// TwinCAT 3 PLC project TestHarnessCore
// Title: TestHarnessCore
// Company: None
// ProjectVersion: 0.0.11
// ProgramVersion: 3.1.4026.24
// libraries:
//   Tc2_Standard, * (Beckhoff Automation GmbH)
//   Tc2_System, * (Beckhoff Automation GmbH)
//   Tc2_Utilities, * (Beckhoff Automation GmbH)
//   Tc3_EventLogger, * (Beckhoff Automation GmbH)
//   Tc3_JsonXml, * (Beckhoff Automation GmbH)
// project tree:
//   DUTs/ E_FailureKind.TcDUT, E_PhaseOutcome.TcDUT, E_RegistrationFault.TcDUT, E_RunOutcome.TcDUT, E_RunPhase.TcDUT, E_TestStatus.TcDUT, ST_CompareResult.TcDUT, ST_NumericValue.TcDUT, ST_TestBudget.TcDUT, ST_TestBudgets.TcDUT, ST_TestRunStatus.TcDUT, ST_TestSlot.TcDUT
//   Interfaces/ I_TestCyclic.TcIO, I_Labelled.TcIO, I_Test.TcIO, I_TestAssertions.TcIO, I_TestConfiguration.TcIO, I_TestDefaults.TcIO, I_TestDetailSink.TcIO, I_TestExecution.TcIO, I_TestJournalSet.TcIO, I_TestLocation.TcIO, I_TestOutcome.TcIO, I_TestRegistrar.TcIO, I_TestReporter.TcIO, I_TestReRun.TcIO, I_TestRegistration.TcIO, I_TestRoster.TcIO, I_TestRunRegistration.TcIO, I_TestRunStatus.TcIO, I_TestSetup.TcIO, I_TestSuite.TcIO, I_TestTeardown.TcIO, I_TestTiming.TcIO
//   Parameters/ TestHarnessParameter.TcGVL
//   POUs/ TestArbiter.TcPOU, TestDeadline.TcPOU, TestEventReporter.TcPOU, TestJournal.TcPOU, TestJUnitReporter.TcPOU, TestLogReporter.TcPOU, TestRegistry.TcPOU, TestReporterFanout.TcPOU, TestRun.TcPOU, TestRunner.TcPOU, TestRunTally.TcPOU, TestStopwatch.TcPOU, TestSuite.TcPOU, TestSummaryLine.TcPOU, TestTimeoutDiagnostic.TcPOU, TestValueAsLReal.TcPOU, TestValueBrief.TcPOU, TestValueCompare.TcPOU, TestValueIsFloat.TcPOU, TestValueIsText.TcPOU, TestValueString.TcPOU, TestVerdict.TcPOU
//   Project Information/ F_GetCompany.TcPOU, F_GetTitle.TcPOU, F_GetVersion.TcPOU
//   Version/ Global_Version.TcGVL
// real-time tasks:
//   TASK PlcTask: cycle T#10ms, priority 20, ADS port 350

// ---- DUTs/E_FailureKind.TcDUT
// Why a test did not pass. Carried in the result document's failure 'type'

// attribute. A single hardcoded 'AssertionError' for everything makes that field

// making a machine-readable field useless.

//

// Keeping the kind here frees the 80-character summary from repeating it, and

// gives CI something to group by.
{attribute 'qualified_only'}
{attribute 'strict'}
TYPE E_FailureKind : (
		None		  := 0,
		ValueMismatch := 1,
		TypeMismatch  := 2,
		SizeMismatch  := 3,
		Timeout		  := 4,
		Aborted		  := 5,
		Environment	  := 6
	) DINT;
END_TYPE

// ---- DUTs/E_PhaseOutcome.TcDUT
// What one scan of TestRunner.Advance did.

//

// TeardownOverran is separate from Finished because the two need different action

// from the caller, and the runner cannot take it: the suite holds the reporters.

// The test's VERDICT is unaffected either way - a passing test whose cleanup hung

// still proved the code correct - but the run must go red, and only the suite can

// say so.
{attribute 'qualified_only'}
{attribute 'strict'}
TYPE E_PhaseOutcome : (
		// Nothing is loaded. Load a test before advancing.
		Idle := 0,
		// Still working. Call again next scan.
		Running := 1,
		// Terminal, cleanly. The verdict is in the journal.
		Finished := 2,
		// Terminal, but teardown hit its deadline and was abandoned. On a rig this may

		// mean an axis left powered. Raise a framework error; do not touch the verdict.
		TeardownOverran := 3
	) DINT;
END_TYPE

// ---- DUTs/E_RegistrationFault.TcDUT
// Why a registration was refused. None means it was accepted.

//

// Distinct causes rather than one BOOL, because each needs a different action from

// whoever reads the report: resize the suite, rename a test, supply the missing

// argument, move the call earlier. A rejected registration is never silent - a

// test that failed to register would otherwise vanish from the results and CI

// would see fewer passes rather than a failure.
{attribute 'qualified_only'}
{attribute 'strict'}
TYPE E_RegistrationFault : (
		None := 0,
		// No free slot. A sizing error: raise the generic argument on the declaration,

		// or split the suite.
		Full := 1,
		// The label is already used in this suite. Labels are the key CI trend history

		// is built on, so two tests cannot share one.
		DuplicateLabel := 2,
		// No label supplied. Usually a missing argument at the call site.
		EmptyLabel := 3,
		// No test supplied. Its own cause rather than folded into EmptyLabel, because

		// reporting the wrong one sends the reader to the wrong argument.
		NoTest := 5,
		// The suite has already been enabled. Registration closes then and a re-run does

		// not reopen it: a re-run re-executes the registered set, it does not redefine

		// it.
		Closed := 4
	) DINT;
END_TYPE

// ---- DUTs/E_RunOutcome.TcDUT
// The aggregate state of a suite, or of a sequencer aggregating suites.

//

// The members mirror E_TestStatus but the type is separate on purpose: a run

// outcome is not a test verdict, and a single type would invite passing one where

// the other is meant.

//

// Aggregation rules, applied in order:

//   any Errored          -> Errored     (the run could not be trusted)

//   any Failed           -> Failed

//   all Skipped          -> Skipped

//   otherwise            -> Passed

//

// Errored outranks Failed because a framework or environment problem casts doubt

// on every other result in the run.
{attribute 'qualified_only'}
{attribute 'strict'}
TYPE E_RunOutcome : (
		NotStarted := 0,
		Running	   := 1,
		Passed	   := 2,
		Failed	   := 3,
		Errored	   := 4,
		Skipped	   := 5
	) DINT;
END_TYPE

// ---- DUTs/E_RunPhase.TcDUT
// Which phase of one test the runner is in. Internal to TestRunner - nothing

// outside it needs to know, and exposing it would invite someone to branch on it.
{attribute 'qualified_only'}
{attribute 'strict'}
TYPE E_RunPhase : (
		Idle	 := 0,
		Setup	 := 1,
		Body	 := 2,
		Teardown := 3
	) DINT;
END_TYPE

// ---- DUTs/E_TestStatus.TcDUT
// The state of a single test.

//

// Six members, each earned: the suite needs to know what to run next, the result

// document needs the four terminal values, and CI needs the last two kept out of

// the failure count.

//

// Errored is deliberately distinct from Failed. Failed means an assertion did not

// hold - the code under test was shown to be wrong. Errored means the test could

// not run: a precondition was absent, a target was unreachable. Conflating them

// sends whoever reads the report hunting a defect that is not there.

//

// The order is NOT load-bearing. Ask IsTerminal() rather than comparing ordinals,

// so that adding a member later is not a breaking change.
{attribute 'qualified_only'}
{attribute 'strict'}
TYPE E_TestStatus : (
		NotStarted := 0,
		Running	   := 1,
		Passed	   := 2,
		Failed	   := 3,
		Errored	   := 4,
		Skipped	   := 5
	) DINT;
END_TYPE

// ---- DUTs/ST_CompareResult.TcDUT
// What TestValueCompare found. A value, not a verdict - nothing is recorded until

// a caller decides to record it.
TYPE ST_CompareResult :
	STRUCT
		IsEqual : BOOL;
		// Why not, when IsEqual is FALSE. None when it is TRUE.
		Kind : E_FailureKind;
		// The composed one-line form, for the summary. Each value in it is shortened to

		// a per-value budget, because both of them plus the surrounding words cannot fit

		// in 255 characters and CONCAT cannot build a longer string than that.

		//

		// Never the author's message - the comparison knows nothing about intent.
		Diagnostic : T_MaxString;
		// The values as rendered, in full, each in its own field so neither is cut by

		// the other. Empty when IsEqual, and empty for a failure that has no two values

		// to show - a size mismatch, a type mismatch.

		//

		// A value whose rendering exceeds 255 characters is still cut here. Comparing

		// something that long is what AssertBufferEqual is for.
		Expected : T_MaxString;
		Actual	 : T_MaxString;
	END_STRUCT
END_TYPE

// ---- DUTs/ST_NumericValue.TcDUT
// A number recovered from an ANY, and whether one was there to recover.

//

// IsNumeric is FALSE for strings, structs, arrays and anything else with no

// ordering. Value is 0.0 in that case and must not be read.

//

// This is a return type rather than an output parameter because an output binds

// with => and never positionally, so a caller writing TestValueAsLReal(V, Ok)

// would bind Ok to an input and never see the flag.
{attribute 'pack_mode' := '1'}
TYPE ST_NumericValue :
	STRUCT
		IsNumeric : BOOL;
		Value	  : LREAL;
	END_STRUCT
END_TYPE

// ---- DUTs/ST_TestBudget.TcDUT
// A deadline for one phase of one test, in both units.

//

// The two units are tracked independently. A test naming its own wall-clock

// budget still inherits the suite's scan budget, and the reverse.

//

// ZERO DISABLES. A budget of zero means no deadline for that unit, which is why

// "not specified" needs its own flag and cannot be inferred from the value. The

// two meanings are different and both are needed: a long-running rig test may

// legitimately want no scan budget at all.
TYPE ST_TestBudget :
	STRUCT
		// Scan budget. The reproducible unit - prefer it. Zero disables.
		Cycles : UDINT;
		// FALSE means "not specified here": inherit the suite default at registration,

		// or leave the existing default unchanged when setting defaults.
		IsCyclesSet : BOOL;
		// Wall-clock budget. Varies with jitter across targets. Zero disables.
		Timeout		 : TIME;
		IsTimeoutSet : BOOL;
	END_STRUCT
END_TYPE

// ---- DUTs/ST_TestBudgets.TcDUT
// The three deadlines a test can have, one per phase.

//

// Three rather than one because the phases are not the same kind of work. Setup

// may legitimately be slow - waiting for hardware to answer. Teardown should not

// be: stopping motion and dropping power is near-immediate, and if it is not,

// that is the fault being detected. Giving teardown the body's budget would leave

// an axis powered for the whole of it.

//

// An untouched instance specifies nothing and inherits every suite default, which

// is what the great majority of registrations want. Declare one in the

// composition root and pass it to every Register that has nothing to say.
TYPE ST_TestBudgets :
	STRUCT
		// Bounds I_TestSetup.Setup. Ignored by a test that does not implement it.
		Setup : ST_TestBudget;
		// Bounds I_Test.Run. This is the original deadline, from when a test grew from

		// one scan to many.
		Body : ST_TestBudget;
		// Bounds I_TestTeardown.Teardown. Overrunning it does NOT change the test's

		// verdict - a passing test whose cleanup hung still proved the code correct -

		// but it is reported as a framework error and turns the run red.
		Teardown : ST_TestBudget;
	END_STRUCT
END_TYPE

// ---- DUTs/ST_TestRunStatus.TcDUT
// The same figures I_TestRunStatus exposes, as a plain struct.

//

// Published alongside the interface so ADS, TwinCAT HMI and OPC UA read the run

// as ordinary symbols without RPC. That is the portable path and the one CI

// polls: an interface is not reachable from outside the PLC, and a design that

// exposed neither - the only signals were a file appearing on disk and a line in

// a log, both of which have to be scraped.
TYPE ST_TestRunStatus :
	STRUCT
		Label	: T_MaxString;
		Outcome : E_RunOutcome;
		// Reached a terminal state - NOT "ran everything". A skipped suite is complete.
		IsComplete : BOOL;
		// Once complete, Passed + Failed + Errored + Skipped equals TestCount.
		TestCount	: UDINT;
		PassedCount : UDINT;
		FailedCount : UDINT;
		// Tests that could not run, plus framework errors. Kept apart from FailedCount

		// because a build should react differently: a failure means the code is wrong,

		// an error means the run cannot be trusted.
		ErrorCount	  : UDINT;
		SkippedCount  : UDINT;
		TotalDuration : LREAL;
	END_STRUCT
END_TYPE

// ---- DUTs/ST_TestSlot.TcDUT
// One registered test, as the registry holds it.

//

// The three optional hooks are resolved ONCE, by __QUERYINTERFACE at registration,

// and stored. Querying them per scan would put an interface lookup in cyclic code

// for a result that cannot change - the instance a slot points at is fixed for the

// life of the run.

//

// A hook the test does not implement is a null reference, which is the whole test:

// no base class, no empty method bodies, no flags to keep in step with reality.
TYPE ST_TestSlot :
	STRUCT
		// Null in a slot that was never claimed. This is the "is there a test here"

		// question - never an index compared against a count.
		Test : I_Test;
		// Where this slot sits in registration order, so a holder of the slot can reach

		// the matching journal without carrying a second value alongside it. -1 in an

		// unclaimed slot.
		Index : DINT := -1;
		Label : T_MaxString;
		// Null unless the test implements the corresponding optional interface.
		Setup	 : I_TestSetup;
		Teardown : I_TestTeardown;
		Location : I_TestLocation;
	END_STRUCT
END_TYPE

// ---- Parameters/TestHarnessParameter.TcGVL
// Dials a referencing project can turn from the Library Manager, without editing

// this library.

//

// Everything here is a DEFAULT, not a limit. Capacity is overridable per instance

// as well - TestRegistry<20> - so this is the value a declaration inherits when it

// says nothing.
{attribute 'qualified_only'}
VAR_GLOBAL CONSTANT
	// Tests a suite can hold. Every slot costs its journal whether used or not, so

	// prefer several small suites to one large one.

	//

	// Must be at least 1: ARRAY[0..Capacity - 1] with zero is a compile error, and

	// that is the right outcome. Clamping a zero to one slot would be the same class

	// of silent surprise this library exists to remove.
	Capacity : UDINT := 10;

	// Sinks a suite or sequencer can hold. Not a generic argument: a project

	// attaches the same set of sinks to every suite it owns, so per-instance

	// variation would cost every declaration site a second argument to buy nothing.
	ReporterCapacity : UDINT := 4;

	// Suites a TestRun can hold. A project usually has a handful - unit, motion,

	// I/O - so this is small on purpose, and overridable per instance as a generic

	// argument like Capacity.
	SuiteCapacity : UDINT := 8;

	// Scans a suite may go WITHOUT COMPLETING A TEST before the run abandons it.

	//

	// Not scans since the suite started - that would fire on a slow suite rather

	// than a stuck one. A rig suite waiting on hardware can sit for minutes and be

	// perfectly healthy, but it still finishes its tests one at a time; a stalled one

	// finishes none.

	//

	// Generous on purpose. This is a BACKSTOP: per-test deadlines already bound

	// every test that did not disable them, so the only things left for this to catch

	// are a framework defect and a test that turned its own deadlines off and hung.

	// A single legitimate test that takes longer than this needs it raised.

	//

	// Zero disables it, like every other deadline in this library.
	SuiteWatchdogCycles : UDINT := 60000;
END_VAR

// ---- Version/Global_Version.TcGVL
{attribute 'TcGenerated'}
{attribute 'no-analysis'}
{attribute 'linkalways'}
// This function has been automatically generated from the project information.
VAR_GLOBAL CONSTANT
	{attribute 'const_non_replaced'}
	stLibVersion_TestHarnessCore : ST_LibVersion := (iMajor := 0, iMinor := 0, iBuild := 11, iRevision := 0, nFlags := 0, sVersion := '0.0.11');
END_VAR

// ---- Interfaces/I_TestCyclic.TcIO
// Something with per-scan work.

//

// The bottom of the stack, with IQueryInterface beneath it. Every interface in

// this library reaches IQueryInterface through its own root, so any reference can

// be queried for any other role it plays.
INTERFACE I_TestCyclic EXTENDS __SYSTEM.IQueryInterface

// Called every scan, unconditionally, by whatever owns this object.

//

// The name is the contract. An Execute input would mean a trigger; an Enable

// input would mean held-while-wanted; CyclicLogic means there is no gating

// condition and the caller must not invent one.
METHOD CyclicLogic
END_METHOD

END_INTERFACE

// ---- Interfaces/I_Labelled.TcIO
// Something that carries a human-readable name.

//

// Extracted because a suite needs a label in two unrelated roles - as the thing

// the sequencer drives, and as the thing an observer reads counts from - and

// declaring it twice would let the two drift apart.
INTERFACE I_Labelled EXTENDS __SYSTEM.IQueryInterface

// The name that appears in results. Stable across renames of the underlying

// instance, because it is supplied rather than derived.
PROPERTY Label : T_MaxString
GET
END_GET
END_PROPERTY

END_INTERFACE

// ---- Interfaces/I_Test.TcIO
// A test. Implemented by test code you write - never by the code under test.

//

// One method is the entire framework contract for a test author.

//

// Reaches IQueryInterface so the suite can ask, at registration, whether a test

// also implements I_TestSetup, I_TestTeardown or I_TestLocation. Those three are

// optional and independent: implement none, one, or all, with no empty bodies for

// the ones you do not want. They do not share a base interface because they would

// have to share a method name, and a test implementing two would then collide.
INTERFACE I_Test EXTENDS __SYSTEM.IQueryInterface

// Called by the suite once per scan while this test is the active one, and never

// otherwise. There is no gate to check and no permission to ask: if you were

// called, run.

//

// Return TRUE when there is no more work. A single-scan test returns TRUE on its

// first call; a multi-scan test returns FALSE until its state machine finishes.

// The test declares completion - the framework never infers it from the checks,

// Without it a test can end at its first passing check and report

// green on work it never reached.

//

// Enable is held TRUE while the test should keep running. The suite drops it to

// abandon a test, on reset or re-run. On a falling edge the test returns its own

// state to its starting condition and returns TRUE; the value is otherwise

// ignored in that case.

//

// The verdict is not returned here. It is whatever the checks recorded through

// Test, and it belongs to the runner.
METHOD Run : BOOL
VAR_INPUT
	Enable : BOOL;
	Test   : I_TestAssertions;
END_VAR
END_METHOD

END_INTERFACE

// ---- Interfaces/I_TestAssertions.TcIO
// The handle a test body reports through: the verdict surface, the runner's

// timing, and the built-in comparisons.

//

// Handed to the test on every call. Never held, never stored.

//

// Everything here is a convenience over I_TestOutcome.RecordPass and

// RecordFailure. Domain helpers should take the narrower I_TestOutcome instead -

// they report, they do not need to compare.

//

// There is no WaitUntil. A test that is not finished returns FALSE from Run and is

// called again; waiting is the absence of returning TRUE.
INTERFACE I_TestAssertions EXTENDS I_TestOutcome, I_TestTiming

// As AssertMemEqual, but lengths are compared first and a mismatch is reported

// as SizeMismatch rather than as a difference at some offset.
METHOD AssertBufferEqual
VAR_INPUT
	pExpected	   : POINTER TO BYTE;
	ExpectedLength : UDINT;
	pActual		   : POINTER TO BYTE;
	ActualLength   : UDINT;
	Message		   : T_MaxString;
END_VAR
END_METHOD

// Asserts the test has COMPLETED no more than Cycles scans. Built on

// I_TestTiming.ElapsedCycles, so it needs no bookkeeping from the test.

//

// The scan in progress is not counted - see I_TestTiming.ElapsedCycles. A body

// checking this on its third call is asserting about the two scans that finished,

// not the three it has been called for. Assert it on the scan AFTER the work is

// done, which is where the answer is known anyway:

//

//   IF Sut.IsDone THEN

//       Test.AssertCompletedWithin(2, 'homing took too long');

//       Run := TRUE;

//   END_IF

//

// Opt-in, never a default. A scan budget is a real regression signal on a fixed

// target and noise across a matrix of them.
METHOD AssertCompletedWithin
VAR_INPUT
	Cycles	: UDINT;
	Message : T_MaxString;
END_VAR
END_METHOD

// Compares two values of the same type, including strings and enums.

//

// ANY binds only to an addressable variable. A literal, a property or an inlined

// constant will not compile, so both sides must be copied into variables first.

// A language constraint, not a choice.
METHOD AssertEqual
VAR_INPUT
	Expected : ANY;
	Actual	 : ANY;
	Message	 : T_MaxString;
END_VAR
END_METHOD

METHOD AssertFalse
VAR_INPUT
	Condition : BOOL;
	Message	  : T_MaxString;
END_VAR
END_METHOD

// Actual > Bound. Numeric types only. See AssertEqual on the ANY constraint.
METHOD AssertGreater
VAR_INPUT
	Actual	: ANY;
	Bound	: ANY;
	Message : T_MaxString;
END_VAR
END_METHOD

// Inclusive on both bounds.
METHOD AssertInRange
VAR_INPUT
	Actual	: LREAL;
	Minimum : LREAL;
	Maximum : LREAL;
	Message : T_MaxString;
END_VAR
END_METHOD

// Actual < Bound. Numeric types only. See AssertEqual on the ANY constraint.
METHOD AssertLess
VAR_INPUT
	Actual	: ANY;
	Bound	: ANY;
	Message : T_MaxString;
END_VAR
END_METHOD

// Byte comparison of two regions of equal length. Reports the offset of the

// first difference.
METHOD AssertMemEqual
VAR_INPUT
	pExpected : POINTER TO BYTE;
	pActual	  : POINTER TO BYTE;
	Length	  : UDINT;
	Message	  : T_MaxString;
END_VAR
END_METHOD

// ABSOLUTE tolerance: passes when |Expected - Actual| <= Tolerance.

//

// Tolerance carries the units of the value compared - millimetres, volts, counts.

// Its counterpart is AssertWithin, which takes a fraction instead.

//

// AssertEqual compares floats EXACTLY. Tolerance is never applied implicitly, so

// choosing it is visible at the call site.
METHOD AssertNear
VAR_INPUT
	Expected  : LREAL;
	Actual	  : LREAL;
	Tolerance : LREAL;
	Message	  : T_MaxString;
END_VAR
END_METHOD

// See AssertEqual on the ANY constraint.
METHOD AssertNotEqual
VAR_INPUT
	Expected : ANY;
	Actual	 : ANY;
	Message	 : T_MaxString;
END_VAR
END_METHOD

METHOD AssertTrue
VAR_INPUT
	Condition : BOOL;
	Message	  : T_MaxString;
END_VAR
END_METHOD

// RELATIVE tolerance: passes when |Expected - Actual| <= |Expected| * Fraction.

//

// Holds its meaning across magnitudes, which absolute tolerance does not. Near

// zero it collapses to exact equality - if zero is the expected value, use

// AssertNear.
METHOD AssertWithin
VAR_INPUT
	Expected : LREAL;
	Actual	 : LREAL;

	// Dimensionless. 0.001 is 0.1 per cent of Expected.
	Fraction : LREAL;
	Message	 : T_MaxString;
END_VAR
END_METHOD

END_INTERFACE

// ---- Interfaces/I_TestConfiguration.TcIO
// Startup configuration common to a suite and a sequencer: what it is called, and

// where its results go. Held by the composition root and nothing else.

//

// Shared by both because both implement I_TestRunStatus - so both carry a label -

// and both fan results out to sinks. The two suite-only faces stay separate:

// I_TestRegistration adds tests, I_TestDefaults sets deadline defaults, and a

// sequencer has neither.

//

// Everything here is set before the object is first enabled. Nothing on this

// interface is safe to call from cyclic code.
INTERFACE I_TestConfiguration EXTENDS __SYSTEM.IQueryInterface

// Attach a sink. Every reporter attached receives every result; there is no

// filtering here, because a sink that wants less can decide that for itself.

//

// Order of attachment is order of notification, which matters for one thing only:

// a sink that writes a file and a sink that raises an alarm should not be relied

// on to complete in any particular order relative to each other. If sequencing

// between two sinks matters, that is one sink wrapping two.

//

// Returns FALSE when the reporter list is full or the object is already running,

// and raises a framework error through the reporters ALREADY attached. That is

// not circular: the ones already there are exactly the ones that can still report

// it. A rejection with no reporters attached at all is silent, and is the reason

// ReporterCount exists.
METHOD AddReporter : BOOL
VAR_INPUT
	Reporter : I_TestReporter;
END_VAR
END_METHOD

// Assert this in CI against an expected number.

//

// A reporter that silently stops being attached takes its output with it - the

// result file simply never appears - and the pipeline reads that as a broken

// build rather than as a missing sink. Same regression hazard as

// I_TestRegistration.RegisteredCount, same mitigation.
PROPERTY ReporterCount : UDINT
GET
END_GET
END_PROPERTY

// What this suite or sequencer is called in the results.

//

// Supplied rather than derived, unlike a test name. A suite is declared once in a

// composition root that is read as configuration, so the label sits where a reader

// is already looking; and the argument for deriving test names - that renaming an

// instance must not silently rename the reported thing - cuts the other way here,

// because CI trend history is grouped by suite and a suite label should survive

// the instance being moved.

//

// An empty label at the point the run starts is a framework error, not an unnamed

// suite in the result document.
METHOD SetLabel
VAR_INPUT
	Label : T_MaxString;
END_VAR
END_METHOD

END_INTERFACE

// ---- Interfaces/I_TestDefaults.TcIO
// Suite-wide deadline defaults, set once at startup alongside registration.

//

// Separate from execution because it has a different holder and a different

// lifetime: the composition root configures, the sequencer drives.

//

// One method rather than six. Three phases times two units is six numbers, and

// six setters would be six chances to set the wrong one; the struct names every

// field at the call site.
INTERFACE I_TestDefaults EXTENDS __SYSTEM.IQueryInterface

// The budgets every test inherits for any phase and unit it did not claim for

// itself at registration.

//

// A field with its IsSet flag FALSE leaves that default as it was, so a caller can

// set the teardown default without restating the other two.

//

// Deadlines are ON by default. An opt-in deadline protects only the tests whose

// authors considered hanging, and those are not the tests that hang. Zero in a

// field that IS set disables that unit deliberately.

//

// Must be called before the suite is first enabled. Defaults are applied to the

// registered set when the run starts; changing them afterwards changes nothing.
METHOD SetDefaults
VAR_INPUT
	Defaults : ST_TestBudgets;
END_VAR
END_METHOD

END_INTERFACE

// ---- Interfaces/I_TestDetailSink.TcIO
// Optional face of a reporter: every check as it is recorded, rather than a

// summary once the test is over.

//

// Discovered with __QUERYINTERFACE on I_TestReporter. A sink that only wants

// verdicts - the event logger, an alarm block - does not implement this and is

// never called for checks.

//

// It exists because the detailed report has no fixed upper size and so cannot be

// a value the framework accumulates. A single comparison of two 255-character

// values already overflows a T_MaxString, and a test may record dozens of checks.

// Buffering that per test would cost the buffer times the suite capacity and

// would still truncate. Streaming costs one buffer per sink that wants one, and

// truncates nothing.

//

// Ordering is guaranteed: TestStarted, then every check in the order the test

// recorded them, then I_TestReporter.TestFinished for the same test. Checks

// recorded during setup and teardown are included, and arrive between the same

// two calls.

//

// These are called from inside the test's own scan. Do the same as any other

// reporter method does with slow work: start it here, advance it in CyclicLogic.
INTERFACE I_TestDetailSink EXTENDS __SYSTEM.IQueryInterface

// One check that did not hold.

//

// Every failure arrives here, including the ones the summary discards: the

// journal keeps only the first for its 80-character line, and this is where the

// rest survive.

//

// Kind and Diagnostic are generated; Message is the author's words, in full and

// never shortened. StepLabel is the label current when the check ran, or empty.

//

// Expected and Actual carry the compared values in full, each in its own field,

// and are empty for a failure that has no two values to show. Diagnostic holds

// the same values shortened to fit one line - so a sink that wants the full text

// composes it from Expected and Actual rather than from Diagnostic.
METHOD CheckFailed
VAR_INPUT
	StepLabel  : T_MaxString;
	Kind	   : E_FailureKind;
	Expected   : T_MaxString;
	Actual	   : T_MaxString;
	Diagnostic : T_MaxString;
	Message	   : T_MaxString;
END_VAR
END_METHOD

// One satisfied check.

//

// Detail is whatever context the caller passed to RecordPass and is usually

// empty. Step is the label current when the check ran, or empty.
METHOD CheckPassed
VAR_INPUT
	StepLabel : T_MaxString;
	Detail	  : T_MaxString;
END_VAR
END_METHOD

// A test has become the active one. Checks for it follow.

//

// Needed because checks now arrive before the test has a verdict, so a sink

// building a document has nowhere to put them unless it is told when to open the

// element. Location is empty if the test does not implement I_TestLocation.
METHOD TestStarted
VAR_INPUT
	SuiteLabel : T_MaxString;
	TestLabel  : T_MaxString;
	Location   : T_MaxString;
END_VAR
END_METHOD

END_INTERFACE

// ---- Interfaces/I_TestExecution.TcIO
// What the sequencer needs to drive a suite, and nothing more.
INTERFACE I_TestExecution EXTENDS __SYSTEM.IQueryInterface

// Called once per scan by the sequencer. Returns TRUE when every registered test

// has reached a terminal state.

//

// The first call with Enable TRUE closes registration and starts the run.

// Dropping Enable abandons it: the active test, and any setup or teardown in

// flight, are cancelled.
METHOD Run : BOOL
VAR_INPUT
	Enable : BOOL;
END_VAR
END_METHOD

// Mark every registered test Skipped without running any, and complete. Must be

// called before the suite is first enabled.

//

// The suite still reports IsComplete. A skipped suite that reported otherwise

// would hang any sequencer aggregating it. Skipped tests do not turn a build red.
METHOD Skip
END_METHOD

END_INTERFACE

// ---- Interfaces/I_TestJournalSet.TcIO
// Bulk operations across every registered journal, at the two moments a run has

// them: starting one, and starting it again.

//

// Held by the suite alone. Deliberately not on I_TestRoster - something that only

// reads the set must not be able to clear every verdict in it.
INTERFACE I_TestJournalSet EXTENDS __SYSTEM.IQueryInterface

// Push the suite defaults into every registered journal, filling whatever each

// test did not claim for itself at registration.

//

// Called once when the run starts, not at registration: the defaults may be set

// after some tests are already registered.
METHOD ApplyDefaults
VAR_INPUT
	Defaults : ST_TestBudgets;
END_VAR
END_METHOD

// Clear every verdict and count, keeping the registered set and the budgets each

// test claimed. This is what a re-run does: it re-executes what was registered, it

// does not redefine it.
METHOD ResetAll
END_METHOD

END_INTERFACE

// ---- Interfaces/I_TestLocation.TcIO
// Optional. Supplies the instance path of a test, carried in the result document

// as 'classname' - where to look when the test fails.

//

// Additive, not a replacement. The label passed to Register is the stable key CI

// history is built on and survives renaming or moving the instance; this is the

// diagnostic that says where the instance actually is.

//

// A test not implementing this reports an empty classname; nothing else changes.

//

// Implement by declaring one TestIdentity member and returning its Path. The three

// attributes it needs are all required - reflection on the function block,

// instance-path and noinit on the string - and a missing one is silent: the

// project compiles and the string stays empty.
INTERFACE I_TestLocation EXTENDS __SYSTEM.IQueryInterface

// e.g. 'Project.PLC.UnitTests.AddsTwoNumbers'
PROPERTY Path : T_MaxString
GET
END_GET
END_PROPERTY

END_INTERFACE

// ---- Interfaces/I_TestOutcome.TcIO
// The verdict surface: recording what a check found, and reading what has been

// recorded so far.

//

// This is the narrow type a domain helper should take. AssertAxisAtPosition needs

// to record a pass or a failure and nothing else - it has no use for the built-in

// comparisons, and taking the full assertion interface would suggest otherwise.

//

// RecordPass and RecordFailure are the primitive pair everything else is built on,

// inside this library and outside it. Fail() alone gives no way to record

// a pass, so an external helper had to write AssertTrue(TRUE) - which produced a

// meaningless message when it went wrong.
INTERFACE I_TestOutcome EXTENDS __SYSTEM.IQueryInterface

// Checks recorded so far, passed and failed.

//

// A test that finishes having recorded none is reported as Errored, not Passed. A

// body that checked nothing usually means a branch never ran - a silent false pass

// wearing a green badge.
PROPERTY AssertionCount : UDINT
GET
END_GET
END_PROPERTY

// Fail outright, with no comparison. For a branch that should be unreachable.
METHOD Fail
VAR_INPUT
	Reason : T_MaxString;
END_VAR
END_METHOD

// Record one failed check and set the verdict to Failed. Later checks are still

// evaluated and recorded, but the verdict cannot return to Passed.
METHOD RecordFailure
VAR_INPUT
	Kind : E_FailureKind;

	// The generated part - values, sizes, byte offset. Composed into the summary

	// after the step label and ahead of the author's message.
	Diagnostic : T_MaxString;

	// The author's words. The first element dropped from the summary if it does

	// not fit, and always present in full in the detail.
	Message : T_MaxString;
END_VAR
END_METHOD

// Record one satisfied check. Does not end the test - a test ends when its Run

// method returns TRUE.
METHOD RecordPass
VAR_INPUT
	// Optional context for the detailed report. Never shown in the summary.
	Detail : T_MaxString;
END_VAR
END_METHOD

// The test could not run - a precondition absent, a target unreachable, a route

// missing. Distinct from failing: the code under test was never exercised, so

// reporting this as a failure would send the reader after the wrong thing.
METHOD ReportError
VAR_INPUT
	Reason : T_MaxString;
END_VAR
END_METHOD

// Label the phase the test is currently in. Purely diagnostic, and worth setting

// even in a test with a single check.

//

// Its value shows in a timeout, which is the dominant failure mode for anything

// multi-scan. 'Home: timed out after 5000 cycles' usually ends an investigation;

// 'timed out after 5000 cycles' starts one.
METHOD SetStep
VAR_INPUT
	Label : T_MaxString;
END_VAR
END_METHOD

// Read-only, deliberately. The original exposed a setter, which let a test body

// write its own verdict and corrupt the run.

//

// Worth reading in a teardown body, which runs whatever the outcome and may need

// to behave differently after a failure.
PROPERTY Status : E_TestStatus
GET
END_GET
END_PROPERTY

END_INTERFACE

// ---- Interfaces/I_TestRegistrar.TcIO
// Putting tests into the registry, and shutting the door. Held by the suite, and

// reached only from the suite's own startup face - a test body cannot get here.

//

// One of three faces on TestRegistry, split by audience for the same reason a

// suite has six. This one WRITES; the arbiter and runner hold I_TestRoster and

// cannot.

//

// The registry is the one generic object in the library, so every consumer reaches

// it through an interface: a generic instance cannot be passed by its concrete

// type at all.
INTERFACE I_TestRegistrar EXTENDS __SYSTEM.IQueryInterface

// Registration is over. Called when the suite is first enabled - not after the

// first scan, because a machine project may need several scans to decide what to

// register.

//

// A re-run does not reopen it.
METHOD Close
END_METHOD

// TRUE until Close. A composition root can assert this rather than discover the

// boundary by being refused.
PROPERTY IsOpen : BOOL
GET
END_GET
END_PROPERTY

// Take the next free slot. Returns None on success, or why it was refused.

//

// Order of claiming is order of execution. The optional hooks are resolved here,

// once, so no __QUERYINTERFACE happens in cyclic code.
METHOD TryClaim : E_RegistrationFault
VAR_INPUT
	Test	: I_Test;
	Label	: T_MaxString;
	Budgets : ST_TestBudgets;
END_VAR
END_METHOD

END_INTERFACE

// ---- Interfaces/I_TestReporter.TcIO
// Where results go. A suite or sequencer holds several and calls all of them.

//

// Implementations: the result-document writer, the event logger, an alarm block

// for a persistent HMI-visible failure state, an ADS logger, a metrics writer, and

// an opt-in message box. A build attaches the sinks it wants.

//

// Reporting is configuration, not behaviour. Severity policy, whether an

// individual re-run is recorded, and which destinations exist are all decided by

// what a build attaches, not by anything inside a test.

//

// Extends I_Cyclic because a reporter must not block: anything slow, a file write

// or an ADS call, is started in one of these methods and advanced in CyclicLogic.

//

// A reporter that wants every individual check, not just the verdict, additionally

// implements I_TestDetailSink. It is found with __QUERYINTERFACE, the same way the

// optional test hooks are, so a sink that does not want checks writes no empty

// method bodies for them.
INTERFACE I_TestReporter EXTENDS I_TestCyclic

// The framework itself could not do something: a rejected registration, a suite

// that never progressed, a result document that could not be written.

//

// Never silent, and never reported as a test failure. Source may be empty - some

// of these occur before any suite is running.
METHOD FrameworkError
VAR_INPUT
	Source	: T_MaxString;
	Message : T_MaxString;
END_VAR
END_METHOD

// FALSE while asynchronous work is in flight.

//

// CI must wait for this as well as IsComplete. A run finishing and its result

// document reaching disk are different events, and copying between them yields a

// truncated artifact - which reads as a broken pipeline rather than a finished run.
PROPERTY IsIdle : BOOL
GET
END_GET
END_PROPERTY

// Every suite the sequencer drives has reached a terminal state.

//

// TargetInfo identifies where the run happened - NetId, platform, TwinCAT

// version. Without it a matrix run across several targets produces result

// documents that cannot be told apart.
METHOD RunFinished
VAR_INPUT
	Status	   : I_TestRunStatus;
	TargetInfo : T_MaxString;
END_VAR
END_METHOD

// A run has begun. Raised once, before anything else in it.

//

// The counterpart of I_TestDetailSink.TestStarted, and it exists for the same

// reason: a sink that BUILDS something is told when to open it rather than

// inferring it from the first thing to arrive. The result-document writer creates

// its document here.

//

// It also lets a log sink bracket its output. Failures stream DURING a run and the

// summary comes at the end, so a marker only at the end would bracket nothing.
METHOD RunStarted
VAR_INPUT
	Label	   : T_MaxString;
	TargetInfo : T_MaxString;
END_VAR
END_METHOD

// One suite reached a terminal state. Status carries the label and the counts.
METHOD SuiteFinished
VAR_INPUT
	Status : I_TestRunStatus;
END_VAR
END_METHOD

// One test reached a terminal state.

//

// Summary is composed to fit 80 characters in a fixed order: step label, then

// generated diagnostic, then the author's message. The author's message is the

// only element that may be dropped, and it is dropped whole rather than cut

// mid-word.

//

// There is no detailed report here. Detail is streamed check by check through

// I_TestDetailSink, which a reporter implements only if it wants it. A single

// T_MaxString could not carry it: one comparison of two 255-character values

// already exceeds 255, so a per-test buffer would truncate exactly the long values

// worth reading.

//

// Kind belongs in the document's 'type' attribute, which frees Summary from

// repeating it and gives CI something to group by - Timeout, ValueMismatch and

// SizeMismatch are different questions and group separately.
METHOD TestFinished
VAR_INPUT
	SuiteLabel : T_MaxString;
	TestLabel  : T_MaxString;

	// Instance path, or empty if the test does not implement I_TestLocation.
	Location	  : T_MaxString;
	Status		  : E_TestStatus;
	Kind		  : E_FailureKind;
	Summary		  : T_MaxString;
	ElapsedTime	  : LREAL;
	ElapsedCycles : UDINT;
	Assertions	  : UDINT;
END_VAR
END_METHOD

END_INTERFACE

// ---- Interfaces/I_TestReRun.TcIO
// Re-execution, for someone at a keyboard. Separate because it is a debugging

// surface, not something CI or the sequencer should hold.
INTERFACE I_TestReRun EXTENDS __SYSTEM.IQueryInterface

// Re-execute every registered test. Clears verdicts and counts and produces a

// fresh result document.
METHOD ReRun
END_METHOD

// Re-execute one test by label. Records no result and writes no document, so a

// session at the keyboard cannot pollute the CI artifact with duplicate entries.

//

// Returns FALSE if the label is not registered.
METHOD ReRunSingle : BOOL
VAR_INPUT
	Label : T_MaxString;
END_VAR
END_METHOD

END_INTERFACE

// ---- Interfaces/I_TestRegistration.TcIO
// The startup-only face of a suite. Held by the composition root and nothing else.

//

// Separated from the driving surface so cyclic code cannot reach Register. A test

// body registering another test mid-run would corrupt the ordering, the counts and

// the statistics, and the sequencer has no reason to see it.
INTERFACE I_TestRegistration EXTENDS __SYSTEM.IQueryInterface

// TRUE until the suite is first enabled. Registration is open until then, not

// merely for the first scan - a machine project may need several scans to decide

// what to register, for instance based on which hardware answered.

//

// A re-run does not reopen it. A re-run re-executes the registered set; it does

// not redefine it.
PROPERTY IsOpen : BOOL
GET
END_GET
END_PROPERTY

// Add a test. Order of registration is order of execution.

//

// The label is required and becomes the result document's 'name' - the key CI

// trend history is built on, so it should read as a description rather than an

// identifier. For an array of parameterised tests, build it:

// CONCAT('Scaling case ', INT_TO_STRING(i)).

//

// Returns FALSE, and raises a framework error naming the label, when the suite is

// full, the label is already used, the label is empty, or registration has closed.

//

// Never silent. A test that failed to register would otherwise vanish from the

// results and CI would see fewer passes rather than a failure - the regression

// hazard RegisteredCount exists to catch.
METHOD Register : BOOL
VAR_INPUT
	Test  : I_Test;
	Label : T_MaxString;

	// This test's own deadlines. An untouched instance claims nothing and inherits

	// every suite default, which is what most registrations want - declare one in

	// the composition root and pass the same one to all of them.

	//

	// Registration is where a deadline is set because it is the only point that is

	// unambiguously before every phase runs. Setup happens before the test's first

	// cycle, so a test cannot set its own setup budget from inside itself; and a

	// budget that could be written from the test body could be moved during the

	// work it bounds.
	Budgets : ST_TestBudgets;
END_VAR
END_METHOD

// Assert this in CI against an expected number. A test that silently stops being

// registered reduces the count, and no other signal exists.
PROPERTY RegisteredCount : UDINT
GET
END_GET
END_PROPERTY

END_INTERFACE

// ---- Interfaces/I_TestRoster.TcIO
// Reading the registered set. What the arbiter and the runner hold, and all they

// hold: neither can register a test, close the window or reset a verdict.

//

// Count lives here rather than on I_TestRegistrar because two interfaces declaring

// one member is a design error even when the types match - the mistake already

// made once in this library with Duration, and corrected in UPDATE_1. The suite

// needs the count too, and reaches it through this face like everyone else.
INTERFACE I_TestRoster EXTENDS __SYSTEM.IQueryInterface

// Tests registered. Assert this in CI against an expected number: a test that

// silently stops being registered reduces it, and no other signal exists.
PROPERTY Count : UDINT
GET
END_GET
END_PROPERTY

// The record for the test at this index, as a reference the runner writes through

// and TestVerdict is retargeted to.

//

// A REFERENCE TO, not a copy: a journal is written continuously while its test

// runs, and a copy would record into something nobody reads. That an interface can

// declare this and that it stays live was probed before being relied on.

//

// An index outside the registered range returns an invalid reference. Check it

// with __ISVALIDREF before use.
METHOD Journal : REFERENCE TO TestJournal
VAR_INPUT
	Index : DINT;
END_VAR
END_METHOD

// Index of the test carrying this label, or -1 if there is none. What

// ReRunSingle resolves a label with.

//

// Not named Find or IndexOf: FIND is a standard string function and INDEXOF is an

// operator, and TwinCAT is case-insensitive.
METHOD Lookup : DINT
VAR_INPUT
	Label : T_MaxString;
END_VAR
END_METHOD

// The registered test at this index, with its label and its resolved hooks.

//

// An index outside the registered range returns an empty slot - a null Test and an

// Index of -1 - rather than faulting, so a caller that has miscounted gets

// something it can test rather than an out-of-bounds read.
METHOD Slot : ST_TestSlot
VAR_INPUT
	Index : DINT;
END_VAR
END_METHOD

END_INTERFACE

// ---- Interfaces/I_TestRunRegistration.TcIO
// Adding suites to a run. The composition root holds this and nothing else does.

//

// Separate from the driving surface for the reason every face in this library is:

// something that only drives a run must not be able to change what is in it, and

// cyclic code must not be able to reach this at all.
INTERFACE I_TestRunRegistration EXTENDS __SYSTEM.IQueryInterface

// Add a suite. Order of addition is order of execution, which is where coarse

// exclusion comes from: two suites touching the same axis cannot overlap because

// only one is ever enabled.

//

// Returns FALSE, and raises a framework error, when the run is full, the suite is

// null, or the run has already started. Never silent - a suite that failed to be

// added takes all its tests with it, and the totals simply come out smaller.
METHOD AddSuite : BOOL
VAR_INPUT
	Suite : I_TestSuite;
END_VAR
END_METHOD

// Assert this in CI against an expected number, for the same reason

// I_TestRegistration.RegisteredCount exists one level down.
PROPERTY SuiteCount : UDINT
GET
END_GET
END_PROPERTY

END_INTERFACE

// ---- Interfaces/I_TestRunStatus.TcIO
// The read model. Implemented by a suite, and by a sequencer aggregating suites -

// which is what makes sequencers nest and lets a consumer poll one symbol

// regardless of how many suites exist.

//

// Read-only, and separate from the driving surface on purpose: something that only

// wants to know whether the run finished should not also be handed the ability to

// restart it.

//

// Computing all of this every scan and exposing none of it is the trap. The counts

// were private and absent from any interface, so nothing could ask whether a run

// had finished - the only signals were a file appearing on disk and a line in a

// log, both of which have to be scraped.

//

// A flat struct carrying the same values is published alongside, so ADS, TwinCAT

// HMI and OPC UA read it as plain symbols without RPC. That is the portable path,

// and the one CI polls.
INTERFACE I_TestRunStatus EXTENDS I_Labelled

// Tests that could not run, plus framework errors. Kept apart from FailedCount

// because a build should react differently: a failure means the code is wrong, an

// error means the run cannot be trusted.
PROPERTY ErrorCount : UDINT
GET
END_GET
END_PROPERTY

// Checks that did not hold.
PROPERTY FailedCount : UDINT
GET
END_GET
END_PROPERTY

// Reached a terminal state - NOT 'ran everything'.

//

// A skipped suite reports complete. If it did not, any aggregate containing one

// would wait for it forever.
PROPERTY IsComplete : BOOL
GET
END_GET
END_PROPERTY

// Readable while the run is in progress, not only at the end: Outcome

// distinguishes Running from every terminal value.
PROPERTY Outcome : E_RunOutcome
GET
END_GET
END_PROPERTY

PROPERTY PassedCount : UDINT
GET
END_GET
END_PROPERTY

// Not a failure. Must not turn a build red.
PROPERTY SkippedCount : UDINT
GET
END_GET
END_PROPERTY

// Tests registered. Once complete, Passed + Failed + Errored + Skipped equals it.
PROPERTY TestCount : UDINT
GET
END_GET
END_PROPERTY

// Seconds for the whole run: a suite sums its tests, a sequencer sums its

// suites.

//

// Named apart from I_TestTiming.ElapsedTime deliberately. The two are not one

// concept declared twice - one is how long a single test has been going, the

// other an aggregate over many. Two interfaces declaring the same member is a

// design error even when the types match, and here the meanings differ too.
PROPERTY TotalDuration : LREAL
GET
END_GET
END_PROPERTY

END_INTERFACE

// ---- Interfaces/I_TestSetup.TcIO
// Optional. Implement when a test needs preparation that may span scans and is

// worth separating from the body.

//

// The suite calls Setup to completion before the first call to Run. A failure or

// error recorded during setup ends the test without running the body - which is

// the point: a test whose fixture never came up has not been exercised, and

// reporting it as a failed check would be a lie.

//

// I_TestTiming.IsFirstCycle covers anything simpler than this.
INTERFACE I_TestSetup EXTENDS __SYSTEM.IQueryInterface

// Return TRUE when setup is complete. Enable behaves as in I_Test.Run.

//

// Bounded by its own deadline, separate from the test's.
METHOD Setup : BOOL
VAR_INPUT
	Enable : BOOL;
	Test   : I_TestAssertions;
END_VAR
END_METHOD

END_INTERFACE

// ---- Interfaces/I_TestSuite.TcIO
// A suite as the sequencer sees it: something to drive, and something to read

// counts from. It adds nothing of its own - it exists so the sequencer can hold

// one reference instead of two that must be kept pointing at the same object.

//

// The other faces of a suite are deliberately not here. I_TestRegistration,

// I_TestDefaults and I_TestConfiguration belong to the composition root,

// I_TestReRun to whoever is debugging. One object, six interfaces, three holders -

// and cyclic code cannot reach registration.
INTERFACE I_TestSuite EXTENDS I_TestExecution, I_TestRunStatus

END_INTERFACE

// ---- Interfaces/I_TestTeardown.TcIO
// Optional. Implement when a test leaves something that must be put back -

// motion stopped, power dropped, a handle closed, a route released.

//

// The suite calls Teardown after the test reaches a verdict, whatever that verdict

// is: passed, failed, errored, timed out or abandoned. This is the guarantee the

// original could not make, because it never called the tests and so could not call

// anything after them.

//

// Read Status if the cleanup differs by outcome. Checks recorded here are

// recorded, but the verdict is already set and they cannot change it.
INTERFACE I_TestTeardown EXTENDS __SYSTEM.IQueryInterface

// Return TRUE when teardown is complete. Enable behaves as in I_Test.Run.

//

// Bounded by its own deadline, and it must be. A test that failed by hanging is

// now being asked to clean up and will most likely hang again - and on a rig that

// means an axis left powered. The suite abandons an overrunning teardown and

// reports it rather than stalling the run.
METHOD Teardown : BOOL
VAR_INPUT
	Enable : BOOL;
	Test   : I_TestAssertions;
END_VAR
END_METHOD

END_INTERFACE

// ---- Interfaces/I_TestTiming.TcIO
// What the runner knows about how long the current test has been going.

//

// Separate from the verdict surface because it has its own consumers: a teardown

// deciding how long to wait, a metrics sink, and AssertCompletedWithin - which is

// built on ElapsedCycles rather than on bookkeeping inside the test.
INTERFACE I_TestTiming EXTENDS __SYSTEM.IQueryInterface

// Scans this test has COMPLETED, counted by the runner.

//

// The reproducible measure. Prefer it to ElapsedTime for anything asserted on.

//

// THE SCAN IN PROGRESS IS NOT COUNTED. The runner ticks the clock after the body

// has run, so a body reading this on its first call sees 0, on its second sees 1,

// and on its Nth sees N-1. That keeps it consistent with IsFirstCycle, which is

// TRUE on the same call this reads 0.

//

// The practical consequence: a body that finishes on its third call must be called

// a third time to observe that it completed two. Establishing that a test finished

// within a budget costs one scan more than the budget - which is cheap, and honest.

// The alternative is a count that includes work not yet done.
PROPERTY ElapsedCycles : UDINT
GET
END_GET
END_PROPERTY

// Seconds elapsed. Wall clock, so it varies with jitter across Windows, BSD,

// Linux RT and containers - report it, but assert on ElapsedCycles.

// Seconds elapsed for this test. Pairs with ElapsedCycles - the same span

// measured two ways.

//

// Wall clock, so it varies with jitter across Windows, BSD, Linux RT and

// containers. Report it; assert on ElapsedCycles.
PROPERTY ElapsedTime : LREAL
GET
END_GET
END_PROPERTY

// TRUE on the first scan of the test body. The setup hook for anything not worth

// implementing I_TestSetup for.
PROPERTY IsFirstCycle : BOOL
GET
END_GET
END_PROPERTY

END_INTERFACE

// ---- POUs/TestRegistry.TcPOU
// The registered set: which tests, in what order, under what labels, with their

// journals.

//

// It exists so the capacity bound lives in ONE place. Expressing the

// same bound as a loop limit in four, and a version existed where ReRunTests

// looped to a parameter while the array was sized by the generic - so a smaller

// instance wrote past the end of its own array. Overflow here is "no free slot

// found", never an index compared against a maximum.

//

// ARRAY[0..Capacity - 1] holds exactly Capacity tests. Declaring

// ARRAY[0.._MaxTestCount], giving N+1, which the README had to explain and which

// leaked into a diagnostic that was simply false.

//

// Capacity must be at least 1. ARRAY[0..-1] is a compile error and that is the

// right outcome - clamping a zero to one slot would be the same class of silent

// surprise this library exists to remove.

//

// THE ONLY GENERIC OBJECT that consumers touch, and the reason every one of them

// touches it through an interface: a generic instance cannot be passed by its

// concrete type, even to something declaring that same type from the same scope.

// Three faces, three audiences - the suite writes, the arbiter and runner read,

// the suite alone resets.
FUNCTION_BLOCK TestRegistry
VAR_GENERIC CONSTANT
	Capacity : UDINT := TestHarnessParameter.Capacity;
END_VAR IMPLEMENTS I_TestRegistrar, I_TestRoster, I_TestJournalSet
VAR
	_Slots : ARRAY[0..Capacity - 1] OF ST_TestSlot;

	// One per slot, sized by the same bound. Separate from ST_TestSlot because a

	// journal is a function block with methods, and the slot is a value.
	_Journals : ARRAY[0..Capacity - 1] OF TestJournal;
	_Count	  : UDINT;
	_IsOpen	  : BOOL := TRUE;

	// Never written. Returned for an out-of-range index so the caller gets a

	// well-defined empty slot rather than whatever was nearby.
	_EmptySlot : ST_TestSlot;
END_VAR

(*
	No cyclic body. The registry is written at startup and read while the run is in
	progress; nothing here has per-scan work.
*)

METHOD ApplyDefaults
VAR_INPUT
	Defaults : ST_TestBudgets;
END_VAR

VAR
	i : DINT;
END_VAR
FOR i := 0 TO TO_DINT(_Count) - 1 DO
	_Journals[i].ApplyDefaults(Defaults);
END_FOR
END_METHOD

METHOD Close
_IsOpen := FALSE;
END_METHOD

PROPERTY Count : UDINT
GET
Count := _Count;
END_GET
END_PROPERTY

PROPERTY IsOpen : BOOL
GET
IsOpen := _IsOpen;
END_GET
END_PROPERTY

METHOD Journal : REFERENCE TO TestJournal
VAR_INPUT
	Index : DINT;
END_VAR
// Invalidated first. A method returning REFERENCE TO that simply returns leaves

// the reference undefined, and undefined reads as valid often enough to pass by
// luck rather than by design.
Journal REF= 0;
IF (Index < 0) OR (Index >= TO_DINT(_Count)) THEN
	RETURN;
END_IF

Journal REF= _Journals[Index];
END_METHOD

METHOD Lookup : DINT
VAR_INPUT
	Label : T_MaxString;
END_VAR

VAR
	i : DINT;
END_VAR
Lookup := -1;
IF Label = '' THEN
	RETURN;
END_IF

// Linear, and deliberately so: it runs at registration and on an individual

// re-run, never per scan, and a sorted structure would cost ordering - which IS

// the execution order.
FOR i := 0 TO TO_DINT(_Count) - 1 DO
	IF _Slots[i].Label = Label THEN
		Lookup := i;
		RETURN;
	END_IF
END_FOR
END_METHOD

METHOD ResetAll
VAR
	i : DINT;
END_VAR
FOR i := 0 TO TO_DINT(_Count) - 1 DO
	_Journals[i].Reset();
END_FOR
END_METHOD

METHOD Slot : ST_TestSlot
VAR_INPUT
	Index : DINT;
END_VAR
// An out-of-range index yields the empty slot: a null Test and an Index of -1.
Slot := _EmptySlot;
IF (Index < 0) OR (Index >= TO_DINT(_Count)) THEN
	RETURN;
END_IF

Slot := _Slots[Index];
END_METHOD

METHOD TryClaim : E_RegistrationFault
VAR_INPUT
	Test	: I_Test;
	Label	: T_MaxString;
	Budgets : ST_TestBudgets;
END_VAR

VAR
	Index : DINT;
END_VAR
IF NOT _IsOpen THEN
	TryClaim := E_RegistrationFault.Closed;
	RETURN;
END_IF

IF Test = 0 THEN
	TryClaim := E_RegistrationFault.NoTest;
	RETURN;
END_IF

IF Label = '' THEN
	TryClaim := E_RegistrationFault.EmptyLabel;
	RETURN;
END_IF

IF THIS^.Lookup(Label) >= 0 THEN
	TryClaim := E_RegistrationFault.DuplicateLabel;
	RETURN;
END_IF

IF _Count >= Capacity THEN
	TryClaim := E_RegistrationFault.Full;
	RETURN;
END_IF

Index				:= TO_DINT(_Count);
_Slots[Index].Test	:= Test;
_Slots[Index].Index := Index;
_Slots[Index].Label := Label;
// Resolved once. A hook the test does not implement stays null, and null is the

// whole mechanism - there is nothing for a test author to opt out of.
IF NOT __QUERYINTERFACE(Test, _Slots[Index].Setup) THEN
	_Slots[Index].Setup := 0;
END_IF

IF NOT __QUERYINTERFACE(Test, _Slots[Index].Teardown) THEN
	_Slots[Index].Teardown := 0;
END_IF

IF NOT __QUERYINTERFACE(Test, _Slots[Index].Location) THEN
	_Slots[Index].Location := 0;
END_IF

_Journals[Index].SetBudgets(Budgets);
_Count	 := _Count + 1;
TryClaim := E_RegistrationFault.None;
END_METHOD

END_FUNCTION_BLOCK

// ---- POUs/TestJournal.TcPOU
// The runner's record of one test: its verdict, its counts, its clock and its

// deadline. One per registered test, owned by the suite.

//

// Written through TestVerdict, read by the reporters. It holds no assertion logic

// and no comparison logic - mixing those in is what takes an object past 673

// lines and made it impossible to test any part of it in isolation.

//

// It holds no detailed report either. Individual checks are streamed to

// I_TestDetailSink as they are recorded; only what the 80-character summary needs

// is kept here, and it is composed once at completion rather than on every check.

// A test with 40 passing checks composes one line and stores nothing per check.
FUNCTION_BLOCK TestJournal
VAR
	_Label	   : T_MaxString;
	_Location  : T_MaxString;
	_Status	   : E_TestStatus;
	_Kind	   : E_FailureKind;
	_StepLabel : T_MaxString;

	// The first failure is kept, not the last. A later failure is usually a

	// consequence of the first, and the first is what the reader must fix.
	_FailDiagnostic : T_MaxString;
	_FailMessage	: T_MaxString;
	_FailStep		: T_MaxString;
	_Summary		: T_MaxString;
	_PassCount		: UDINT;
	_FailCount		: UDINT;
	_ElapsedCycles	: UDINT;
	_IsFirstCycle	: BOOL;

	// All three phases. Only Body is enforced here - the runner bounds the other

	// two, which run outside the span this object measures.
	_Budgets   : ST_TestBudgets;
	_Stopwatch : TestStopwatch;
END_VAR

(*
	No cyclic body. The suite calls Tick once per scan for the active test; every
	other entry point is driven by a recorded check.
*)

// Suite-wide budgets, applied to every phase and unit the test did not claim for

// itself at registration.

//

// Each unit is tracked separately on purpose. A test naming its own wall-clock

// budget still inherits the suite's scan budget, and the reverse. A single

// 'overridden' flag would break exactly that case and nothing else would notice.

//

// Called once, when the run starts. The defaults are not re-applied on a re-run:

// what a test claimed at registration it keeps.
METHOD ApplyDefaults
VAR_INPUT
	Defaults : ST_TestBudgets;
END_VAR
IF NOT _Budgets.Setup.IsCyclesSet THEN
	_Budgets.Setup.Cycles := Defaults.Setup.Cycles;
END_IF

IF NOT _Budgets.Setup.IsTimeoutSet THEN
	_Budgets.Setup.Timeout := Defaults.Setup.Timeout;
END_IF

IF NOT _Budgets.Body.IsCyclesSet THEN
	_Budgets.Body.Cycles := Defaults.Body.Cycles;
END_IF

IF NOT _Budgets.Body.IsTimeoutSet THEN
	_Budgets.Body.Timeout := Defaults.Body.Timeout;
END_IF

IF NOT _Budgets.Teardown.IsCyclesSet THEN
	_Budgets.Teardown.Cycles := Defaults.Teardown.Cycles;
END_IF

IF NOT _Budgets.Teardown.IsTimeoutSet THEN
	_Budgets.Teardown.Timeout := Defaults.Teardown.Timeout;
END_IF
END_METHOD

// Passed and failed together.
PROPERTY AssertionCount : UDINT
GET
AssertionCount := _PassCount + _FailCount;
END_GET
END_PROPERTY

// Called once by the suite when this test becomes the active one.
METHOD Begin
VAR_INPUT
	Label	 : T_MaxString;
	Location : T_MaxString;
END_VAR
THIS^.Reset();
_Label		  := Label;
_Location	  := Location;
_Status		  := E_TestStatus.Running;
_IsFirstCycle := TRUE;
_Stopwatch.Start();
END_METHOD

// The resolved budgets for all three phases, read by the runner to arm the setup

// and teardown deadlines. Valid once the run has started and ApplyDefaults has

// been called.
PROPERTY Budgets : ST_TestBudgets
GET
Budgets := _Budgets;
END_GET
END_PROPERTY

PROPERTY ElapsedCycles : UDINT
GET
ElapsedCycles := _ElapsedCycles;
END_GET
END_PROPERTY

// Seconds elapsed for this test. Backs I_TestTiming.ElapsedTime.
PROPERTY ElapsedTime : LREAL
GET
ElapsedTime := _Stopwatch.Elapsed;
END_GET
END_PROPERTY

// Terminal. Composes the summary once and stops the clock.

//

// Named Finish, not Complete: a status word as a method name reads as a question,

// and

// Complete collides with IsComplete on the status interface.

//

// A Passed verdict with no recorded check becomes Errored: a body that checked

// nothing usually means a branch never ran, and reporting that green is a silent

// false pass.
METHOD Finish
VAR_INPUT
	Status : E_TestStatus;
END_VAR
IF _Status <> E_TestStatus.Running THEN
	RETURN;
END_IF

_Stopwatch.Stop();
IF _FailCount > 0 THEN
	_Status := SEL(_Kind = E_FailureKind.Environment, E_TestStatus.Failed, E_TestStatus.Errored);
ELSIF (Status = E_TestStatus.Passed) AND (_PassCount = 0) THEN
	_Status			:= E_TestStatus.Errored;
	_Kind			:= E_FailureKind.Environment;
	_FailDiagnostic := 'completed without recording a check';
ELSE
	_Status := Status;
END_IF

_Summary := TestSummaryLine(StepLabel := _FailStep, Diagnostic := _FailDiagnostic, Message := _FailMessage);
END_METHOD

PROPERTY IsFirstCycle : BOOL
GET
IsFirstCycle := _IsFirstCycle;
END_GET
END_PROPERTY

PROPERTY Kind : E_FailureKind
GET
Kind := _Kind;
END_GET
END_PROPERTY

PROPERTY Label : T_MaxString
GET
Label := _Label;
END_GET
END_PROPERTY

PROPERTY Location : T_MaxString
GET
Location := _Location;
END_GET
SET
// R13: validated before storing. An instance path is a diagnostic, so a bad one

// should read as "not supplied" rather than send the reader somewhere that does

// not exist.

//

// Length is the only check available: T_MaxString truncates silently at 255, and a

// path cut mid-segment names a place that is not there. An empty classname is
// honest; a wrong one is worse than none.
IF LEN(Location) >= 255 THEN
	_Location := '';
	RETURN;
END_IF

_Location := Location;
END_SET
END_PROPERTY

// Terminal without running. A skipped test is not a failure and must not turn a

// build red.
METHOD MarkSkipped
THIS^.Reset();
_Status := E_TestStatus.Skipped;
END_METHOD

// One failed check. The verdict becomes Failed and cannot return to Passed.

//

// Only the FIRST failure's text is kept for the summary. A later failure is

// usually downstream of the first, and the summary has room for one. Every

// failure, including the discarded ones, still reaches the detail sink.
METHOD RecordFailure
VAR_INPUT
	Kind	   : E_FailureKind;
	Diagnostic : T_MaxString;
	Message	   : T_MaxString;
END_VAR
_FailCount := _FailCount + 1;
IF _FailCount = 1 THEN
	_Kind			:= Kind;
	_FailDiagnostic := Diagnostic;
	_FailMessage	:= Message;
	_FailStep		:= _StepLabel;
END_IF
END_METHOD

// One satisfied check. Nothing but the count: the check's own text goes straight

// to the detail sink and is never held here.
METHOD RecordPass
_PassCount := _PassCount + 1;
END_METHOD

// Back to as-declared, keeping the label and location. Used by a re-run: the

// registered set is not redefined, only re-executed.
METHOD Reset
_Status			:= E_TestStatus.NotStarted;
_Kind			:= E_FailureKind.None;
_StepLabel		:= '';
_FailDiagnostic := '';
_FailMessage	:= '';
_FailStep		:= '';
_Summary		:= '';
_PassCount		:= 0;
_FailCount		:= 0;
_ElapsedCycles	:= 0;
_IsFirstCycle	:= FALSE;
_Stopwatch.Reset();
END_METHOD

// What this test claimed for itself at registration. Whatever it did not claim is

// filled in from the suite defaults when the run starts.

//

// Set once, before anything runs, and never while a phase is in progress. A

// deadline that can move during the work it bounds stops detecting the thing it

// exists for.
METHOD SetBudgets
VAR_INPUT
	Budgets : ST_TestBudgets;
END_VAR
_Budgets := Budgets;
END_METHOD

// Purely diagnostic. Its value is captured with the first failure, so a later

// step cannot relabel an earlier one.
METHOD SetStep
VAR_INPUT
	Label : T_MaxString;
END_VAR
_StepLabel := Label;
END_METHOD

PROPERTY Status : E_TestStatus
GET
Status := _Status;
END_GET
END_PROPERTY

// The step label currently set, or empty. Read by TestVerdict so a streamed check

// carries the step it ran under, and by a teardown that behaves differently

// depending on how far the test got.

//

// Read-only. SetStep is the only way in.
PROPERTY StepLabel : T_MaxString
GET
StepLabel := _StepLabel;
END_GET
END_PROPERTY

// Composed to fit 80 characters. Empty until the test completes.
PROPERTY Summary : T_MaxString
GET
Summary := _Summary;
END_GET
END_PROPERTY

// Advance one scan. Returns TRUE if a deadline has just expired, in which case

// the suite abandons the test - the verdict is already recorded here.

//

// Called AFTER the test body has run, so a budget of one allows one execution.

// That ordering is also why ElapsedCycles reads N-1 during the body's Nth call:

// the scan in progress has not completed, so it is not counted. A test observing

// its own duration needs one scan more than the duration it observes.
METHOD Tick : BOOL
Tick := FALSE;
IF _Status <> E_TestStatus.Running THEN
	RETURN;
END_IF

// Only the first scan is the first scan.
_IsFirstCycle  := FALSE;
_ElapsedCycles := _ElapsedCycles + 1;
IF (_Budgets.Body.Cycles > 0) AND (_ElapsedCycles >= _Budgets.Body.Cycles) THEN
	THIS^.RecordFailure(Kind	   := E_FailureKind.Timeout,
						Diagnostic := TestTimeoutDiagnostic(Phase	 := '',
															Cycles	 := _Budgets.Body.Cycles,
															Timeout	 := _Budgets.Body.Timeout,
															ByCycles := TRUE),
						Message := '');

	THIS^.Finish(E_TestStatus.Failed);
	Tick := TRUE;
	RETURN;
END_IF

IF (_Budgets.Body.Timeout > T#0S) AND (_Stopwatch.Elapsed >= (TO_LREAL(TIME_TO_UDINT(_Budgets.Body.Timeout)) / 1000.0)) THEN
	THIS^.RecordFailure(Kind	   := E_FailureKind.Timeout,
						Diagnostic := TestTimeoutDiagnostic(Phase	 := '',
															Cycles	 := _Budgets.Body.Cycles,
															Timeout	 := _Budgets.Body.Timeout,
															ByCycles := FALSE),
						Message := '');

	THIS^.Finish(E_TestStatus.Failed);
	Tick := TRUE;
END_IF
END_METHOD

END_FUNCTION_BLOCK

// ---- POUs/TestStopwatch.TcPOU
// Elapsed seconds, measured in task scans.

//

// Carried over essentially unchanged - one of the few parts that

// needed nothing. Resolution is the task period, so a test shorter than one scan

// reports zero. That is honest: at this resolution there is nothing finer to say.

//

// Duration is reported, never asserted on. Scan counts are the reproducible

// measure across Windows, BSD, Linux RT and containers.
FUNCTION_BLOCK TestStopwatch
VAR
	_StartCycle		 : UDINT;
	_PreviousElapsed : LREAL;
	_IsRunning		 : BOOL;
END_VAR

(*
	No cyclic body. Elapsed is derived from the task's own cycle counter, so
	nothing has to be called every scan to keep it accurate.
*)

// Seconds since Start, or the frozen value once stopped.
PROPERTY Elapsed : LREAL
GET
VAR
	Cycles : UDINT;
END_VAR
IF NOT _IsRunning THEN
	Elapsed := _PreviousElapsed;
	RETURN;
END_IF

// Unsigned subtraction, so a wrapped cycle counter still yields the correct

// difference.
Cycles := TwinCAT_SystemInfoVarList._TaskInfo[GETCURTASKINDEXEX()].CycleCount - _StartCycle;

// CycleTime is in 100 ns units.
Elapsed := TO_LREAL(Cycles) * TO_LREAL(TwinCAT_SystemInfoVarList._TaskInfo[GETCURTASKINDEXEX()].CycleTime) / 10000000.0;
END_GET
END_PROPERTY

PROPERTY IsRunning : BOOL
GET
IsRunning := _IsRunning;
END_GET
END_PROPERTY

METHOD Reset
_PreviousElapsed := 0.0;
_StartCycle		 := 0;
_IsRunning		 := FALSE;
END_METHOD

// Restarts from zero. Starting an already-running stopwatch discards what it had.
METHOD Start
_PreviousElapsed := 0.0;
_StartCycle		 := TwinCAT_SystemInfoVarList._TaskInfo[GETCURTASKINDEXEX()].CycleCount;
_IsRunning		 := TRUE;
END_METHOD

// Freezes and returns the elapsed seconds. Stopping a stopped stopwatch returns

// what it already held rather than zero.
METHOD Stop : LREAL
IF _IsRunning THEN
	_PreviousElapsed := THIS^.Elapsed;
	_IsRunning		 := FALSE;
END_IF

Stop := _PreviousElapsed;
END_METHOD

END_FUNCTION_BLOCK

// ---- POUs/TestSummaryLine.TcPOU
// Composes the one-line summary that CI list views render.

//

// Pure, and separate from the journal, because the composition rule is worth

// testing on its own - it is the part most likely to be got subtly wrong.

//

// Order is fixed: step label, then generated diagnostic, then the author's

// message. Nothing is cut mid-word. The author's message is the only element that

// may be dropped, and it is dropped whole - it appears in full in the detail

// either way, so a truncated copy in the summary buys nothing and costs

// legibility.

//

// The step label leads because timeout is the dominant failure mode for anything

// multi-scan, and there the label IS the diagnostic: 'Home: timed out after 5000

// cycles' usually ends an investigation.

//

// The failure kind is deliberately absent - it travels in the result document's

// 'type' attribute, where CI can group by it.
FUNCTION TestSummaryLine : STRING
VAR_INPUT
	StepLabel  : T_MaxString;
	Diagnostic : T_MaxString;
	Message	   : T_MaxString;
END_VAR

VAR CONSTANT
	// STRING is STRING(80). Composing to fit is the point of this function.
	MaxLength : INT := 80;
END_VAR

VAR
	Built : T_MaxString;
END_VAR

Built := '';
IF StepLabel <> '' THEN
	Built := CONCAT(StepLabel, ': ');
END_IF

Built := CONCAT(Built, Diagnostic);
// Appended only if the whole of it fits. A partial message is worse than none:

// the reader cannot tell whether the sentence ended or the buffer did.
IF Message <> '' THEN
	IF Built = '' THEN
		IF LEN(Message) <= MaxLength THEN
			Built := Message;
		END_IF
	ELSIF LEN(Built) + 3 + LEN(Message) <= MaxLength THEN
		Built := CONCAT(CONCAT(Built, ' - '), Message);
	END_IF
END_IF

// A diagnostic alone can still overrun - a compared string may be long. Cut it

// with an ellipsis so the reader knows to look at the detail.
IF LEN(Built) > MaxLength THEN
	Built := CONCAT(LEFT(Built, TO_INT(MaxLength - 3)), '...');
END_IF

TestSummaryLine := Built;

END_FUNCTION

// ---- POUs/TestTimeoutDiagnostic.TcPOU
// The one place a deadline expiry is put into words.

//

// Two objects detect timeouts - TestJournal for the body, TestDeadline for setup

// and teardown - and a reader comparing two reports should not have to work out

// whether two differently-worded lines mean the same thing.

//

// Pure, so the wording is testable without running a test that hangs.
FUNCTION TestTimeoutDiagnostic : T_MaxString
VAR_INPUT
	// 'setup', 'teardown', or empty for the test body.
	Phase : T_MaxString;

	// The budget that expired. Only the one named by ByCycles is read.
	Cycles	 : UDINT;
	Timeout	 : TIME;
	ByCycles : BOOL;
END_VAR

IF ByCycles THEN
	TestTimeoutDiagnostic := CONCAT(CONCAT('timed out after ', LREAL_TO_FMTSTR(TO_LREAL(Cycles), 0, FALSE)), ' cycles');
ELSE
	TestTimeoutDiagnostic := CONCAT(CONCAT('timed out after ', TIME_TO_STRING(Timeout)), ' of wall time');
END_IF

IF Phase <> '' THEN
	TestTimeoutDiagnostic := CONCAT(CONCAT(Phase, ' '), TestTimeoutDiagnostic);
END_IF

END_FUNCTION

// ---- POUs/TestRun.TcPOU
// A RUN: the boundary around one or more suites, and the only thing that says a
// run has ended.
//
// It exists because a suite is not a run. RunFinished is a run-level event, and a
// suite raising it would have to know whether anything sits above it. Here the
// answer is structural: a single suite is composed with one TestRun, a sequencer
// IS one, and exactly one object is ever in a position to announce the end.
//
// EVERY PROJECT NEEDS ONE, including a project with a single suite. The result
// document is written on RunFinished, so without a run there is no artifact.
//
// Implements I_TestRunStatus, so runs nest: a consumer polls one symbol regardless
// of how many suites exist, and an outer run absorbs an inner one exactly as this
// absorbs a suite. Counts are TESTS at every level.
//
// A RE-RUN is a run-level operation too, for the same reason: it must produce a
// fresh document, and only this object can announce one.
//
// IT ALSO CARRIES THE SUITE WATCHDOG. A suite that stops progressing cannot see
// that about itself - it is the thing that has stopped - so the object owning the
// sequence is the only one positioned to notice.
//
// Suites run ONE AT A TIME, in the order they were added. That is where coarse
// exclusion comes from - two suites touching the same axis cannot overlap, because
// only one is ever enabled.
FUNCTION_BLOCK TestRun
VAR_GENERIC CONSTANT
	Capacity : UDINT := TestHarnessParameter.SuiteCapacity;
END_VAR IMPLEMENTS I_TestRunRegistration, I_TestConfiguration, I_TestExecution, I_TestRunStatus
VAR
	_Suites : ARRAY[0..Capacity - 1] OF I_TestSuite;
	_Count	: UDINT;
	_Index	: DINT;

	_Tally	: TestRunTally;
	_Fanout : TestReporterFanout;

	// Held so a suite added AFTER a reporter still receives it.
	_Reporters	   : ARRAY[0..TestHarnessParameter.ReporterCapacity - 1] OF I_TestReporter;
	_ReporterCount : UDINT;

	_Label		: T_MaxString;
	_TargetInfo : T_MaxString;
	_IsOpen		: BOOL := TRUE;

	_PendingErrors : UDINT;

	// -- the suite watchdog ----------------------------------------------------
	// Scans the ACTIVE suite has gone without completing a test, and the budget it
	// is measured against.
	_WatchdogCycles : UDINT := TestHarnessParameter.SuiteWatchdogCycles;
	_StallCycles	: UDINT;
	// Verdicts the active suite had reached when it was last seen to progress.
	_LastProgress	: UDINT;
	_StalledSuites	: UDINT;
END_VAR

(*
	No cyclic body. This object is driven through Run, like a suite.
*)

// Attach a sink to the run AND to every suite in it.
//
// One attachment point. A composition root that had to attach the same reporter to
// the run and to each suite separately would eventually miss one, and a suite whose
// results reach no sink is invisible rather than wrong.
METHOD AddReporter : BOOL
VAR_INPUT
	Reporter : I_TestReporter;
END_VAR

VAR
	i : DINT;
END_VAR
AddReporter := FALSE;

IF Reporter = 0 THEN
	RETURN;
END_IF

IF _ReporterCount >= TestHarnessParameter.ReporterCapacity THEN
	THIS^.RaiseFrameworkError('the run cannot hold another reporter');
	RETURN;
END_IF

_Reporters[TO_DINT(_ReporterCount)] := Reporter;
_ReporterCount := _ReporterCount + 1;

_Fanout.Attach(Reporter);

// Suites added before this reporter was.
FOR i := 0 TO TO_DINT(_Count) - 1 DO
	THIS^.PushReporter(_Suites[i], Reporter);
END_FOR

AddReporter := TRUE;
END_METHOD

// Add a suite to the run. Order of addition is order of execution.
//
// That ordering is what gives coarse exclusion for free: two integration suites
// touching the same axis cannot overlap, because only one is ever enabled.
METHOD AddSuite : BOOL
VAR_INPUT
	Suite : I_TestSuite;
END_VAR

VAR
	Index : DINT;
	i	  : DINT;
END_VAR
AddSuite := FALSE;

IF Suite = 0 THEN
	THIS^.RaiseFrameworkError('a null suite was offered');
	RETURN;
END_IF

IF NOT _IsOpen THEN
	THIS^.RaiseFrameworkError('suites cannot be added once the run has started');
	RETURN;
END_IF

IF _Count >= Capacity THEN
	THIS^.RaiseFrameworkError('the run is full - raise its capacity argument');
	RETURN;
END_IF

Index		 := TO_DINT(_Count);
_Suites[Index] := Suite;
_Count		 := _Count + 1;

// Reporters already attached reach this suite too, so the composition root
// attaches once - to the run - whatever order it does things in.
FOR i := 0 TO TO_DINT(_ReporterCount) - 1 DO
	THIS^.PushReporter(Suite, _Reporters[i]);
END_FOR

AddSuite := TRUE;
END_METHOD

// Start the aggregate, and re-apply anything raised before it existed.
//
// A framework error raised while the run was still OPEN - a refused suite, a
// refused reporter - has no tally to record itself into. It is counted in
// _PendingErrors and re-applied here, or a run that could not be composed
// properly reports green with its missing tests simply absent from the totals.
//
// ORDER MATTERS: Begin clears ErrorCount, so the drain must follow it. Both entry
// points into a run go through this method for that reason.
//
// _PendingErrors is NOT cleared. A suite that failed to be added is still missing
// on a re-run, so the error is re-applied every time the aggregate restarts.
METHOD BeginTally
VAR
	i : DINT;
END_VAR
_Tally.Begin(0);

FOR i := 1 TO TO_DINT(_PendingErrors) DO
	_Tally.RecordFrameworkError();
END_FOR
END_METHOD

// Has the active suite stopped making progress?
//
// PROGRESS, not duration. The measure is how many tests the suite has brought to
// a verdict - passed, failed, errored or skipped. A slow suite still moves that
// number; a stalled one does not, and counting scans since it STARTED would fire
// on the slow rather than the stuck.
//
// A suite cannot see this about itself: it is the thing that has stopped. The run
// owns the sequence, so it is the only object positioned to notice.
METHOD CheckWatchdog
VAR_INPUT
	Index : DINT;
END_VAR

VAR
	Progress : UDINT;
	Suite	 : I_TestSuite;
END_VAR
IF _WatchdogCycles = 0 THEN
	RETURN;
END_IF

Suite := _Suites[Index];

IF Suite = 0 THEN
	RETURN;
END_IF

// Every verdict the suite has reached so far.
Progress := Suite.PassedCount + Suite.FailedCount
		  + Suite.ErrorCount + Suite.SkippedCount;

IF Progress <> _LastProgress THEN
	_LastProgress := Progress;
	_StallCycles  := 0;
	RETURN;
END_IF

_StallCycles := _StallCycles + 1;

IF _StallCycles < _WatchdogCycles THEN
	RETURN;
END_IF

// Stalled. Named, counted, and left behind.
_StalledSuites := _StalledSuites + 1;
THIS^.RaiseFrameworkError(CONCAT(CONCAT(
	'suite stalled and was abandoned: ', Suite.Label),
	CONCAT(', no verdict for ', UDINT_TO_STRING(_WatchdogCycles))));

// One call with Enable FALSE, so the suite can put its own state back. Its return
// is ignored: a suite that has stopped will not answer this either, and waiting
// for it would reproduce the stall the watchdog exists to break.
Suite.Run(Enable := FALSE);

// Whatever it did manage still counts.
_Tally.Absorb(Suite);

THIS^.NextSuite();
END_METHOD

PROPERTY ErrorCount : UDINT
GET
ErrorCount := _Tally.ErrorCount;
END_GET
END_PROPERTY

PROPERTY FailedCount : UDINT
GET
FailedCount := _Tally.FailedCount;
END_GET
END_PROPERTY

// Terminal. Settles the aggregate and raises RunFinished - ONCE, whatever the
// topology.
//
// THIS IS WHY THIS OBJECT EXISTS. A suite cannot raise it: a suite is not a run,
// and asking one to announce the end of something above itself is what forced a
// "am I being sequenced" flag in an earlier design. Here a single suite is
// composed with one TestRun and a sequencer IS one, so exactly one object is ever
// in a position to say the run is over.
METHOD Finish
IF _Tally.IsComplete THEN
	RETURN;
END_IF

_Tally.Finish();
_Fanout.RunFinished(Status := THIS^, TargetInfo := _TargetInfo);
END_METHOD

PROPERTY IsComplete : BOOL
GET
IsComplete := _Tally.IsComplete;
END_GET
END_PROPERTY

PROPERTY Label : T_MaxString
GET
Label := _Label;
END_GET
END_PROPERTY

// Move to the next suite and reset the watchdog with it. One place, so the reset
// cannot be forgotten on one of the paths that advances.
METHOD NextSuite
_Index		  := _Index + 1;
_StallCycles  := 0;
_LastProgress := 0;
END_METHOD

PROPERTY Outcome : E_RunOutcome
GET
Outcome := _Tally.Outcome;
END_GET
END_PROPERTY

PROPERTY PassedCount : UDINT
GET
PassedCount := _Tally.PassedCount;
END_GET
END_PROPERTY

// Hand a reporter to a suite through its configuration face.
//
// A suite is held as I_TestSuite - the driving surface - which deliberately does
// not carry AddReporter. The configuration face is reached with __QUERYINTERFACE,
// the same way every optional face in this library is.
METHOD PushReporter
VAR_INPUT
	Suite	 : I_TestSuite;
	Reporter : I_TestReporter;
END_VAR

VAR
	ConfigFace : I_TestConfiguration;
END_VAR
IF Suite = 0 THEN
	RETURN;
END_IF

IF __QUERYINTERFACE(Suite, ConfigFace) THEN
	ConfigFace.AddReporter(Reporter);
END_IF
END_METHOD

// One place run-level framework errors are named.
METHOD RaiseFrameworkError
VAR_INPUT
	Message : T_MaxString;
END_VAR
IF _IsOpen THEN
	// Before the tally exists. Held, and re-applied by BeginTally when the run
	// starts - without that, a run that could not be composed properly reports
	// green with its missing tests simply absent from the totals.
	_PendingErrors := _PendingErrors + 1;
ELSE
	_Tally.RecordFrameworkError();
END_IF

_Fanout.FrameworkError(Source := _Label, Message := Message);
END_METHOD

PROPERTY ReporterCount : UDINT
GET
ReporterCount := _Fanout.Count;
END_GET
END_PROPERTY

// Re-execute every suite in the run, and produce a FRESH document.
//
// It lives here rather than on a suite because the document boundary does. A suite
// re-running on its own re-executes its tests and raises SuiteFinished again, but
// announces no run - so no new artifact is written and the re-run is invisible to
// CI.
//
// The registered set is not redefined, at either level. A re-run re-executes what
// was composed; it does not recompose it.
//
// There is no ReRunSingle here. Re-running ONE thing is a debugging aid scoped to
// a test, and the suite already offers it - a run-level equivalent would be a
// second way to spell the same intention.
METHOD ReRun
VAR
	i		: DINT;
	ReRunFace : I_TestReRun;
END_VAR
IF _IsOpen THEN
	// Never started. There is nothing to repeat.
	RETURN;
END_IF

IF NOT _Tally.IsComplete THEN
	// Mid-run. Restarting now would leave suites half-executed and the counts
	// meaningless.
	THIS^.RaiseFrameworkError('ReRun was called while the run was still going');
	RETURN;
END_IF

FOR i := 0 TO TO_DINT(_Count) - 1 DO
	IF __QUERYINTERFACE(_Suites[i], ReRunFace) THEN
		ReRunFace.ReRun();
	END_IF
END_FOR

// Counts start again from nothing, and Finish will raise RunFinished a second
// time - which is what produces the fresh document. Anything refused at
// composition is re-applied: a suite that never made it in is still missing.
THIS^.BeginTally();
_Index		  := 0;
_StallCycles  := 0;
_LastProgress := 0;
END_METHOD

// Drive the run. One suite at a time, in the order they were added.
//
// Returns TRUE once every suite has reached a terminal state.
METHOD Run : BOOL
VAR_INPUT
	Enable : BOOL;
END_VAR

VAR
	Index : DINT;
END_VAR
_Fanout.CyclicLogic();

Run := _Tally.IsComplete;

IF NOT Enable THEN
	RETURN;
END_IF

IF _IsOpen THEN
	_IsOpen := FALSE;
	THIS^.BeginTally();

	IF _Label = '' THEN
		THIS^.RaiseFrameworkError('the run was started with no label');
	END_IF

	// Once, before anything else in the run. A sink that builds something opens it
	// here rather than guessing from the first result to arrive.
	_Fanout.RunStarted(Label := _Label, TargetInfo := _TargetInfo);
END_IF

IF _Tally.IsComplete THEN
	RETURN;
END_IF

IF _Index >= TO_DINT(_Count) THEN
	THIS^.Finish();
	Run := _Tally.IsComplete;
	RETURN;
END_IF

Index := _Index;

// Serial by construction. Only one suite is ever enabled, which is what makes two
// suites touching the same axis unable to overlap.
IF _Suites[Index].Run(Enable := TRUE) THEN
	// Counts TESTS, not suites, so the figures mean the same thing at every level
	// of a nest.
	_Tally.Absorb(_Suites[Index]);
	THIS^.NextSuite();
ELSE
	THIS^.CheckWatchdog(Index);
END_IF

Run := _Tally.IsComplete;
END_METHOD

METHOD SetLabel
VAR_INPUT
	Label : T_MaxString;
END_VAR
_Label := Label;
_Tally.SetLabel(Label);
END_METHOD

// Where this run happened - NetId, platform, TwinCAT version, whatever
// identifies the machine.
//
// Without it a matrix run across several targets produces result documents that
// cannot be told apart.
METHOD SetTargetInfo
VAR_INPUT
	TargetInfo : T_MaxString;
END_VAR
_TargetInfo := TargetInfo;
END_METHOD

// How many scans a suite may go WITHOUT COMPLETING A TEST before the run
// abandons it. Zero disables the watchdog.
//
// A backstop, not a deadline. Per-test budgets already bound every test that did
// not disable them; this catches what they cannot - a suite that stops progressing
// for any other reason, including a test that turned its own deadlines off.
//
// Raise it for a suite with a single legitimately long test: the count is scans
// between VERDICTS, so one test taking longer than the budget looks identical to
// a suite that has stopped.
METHOD SetWatchdog
VAR_INPUT
	Cycles : UDINT;
END_VAR
_WatchdogCycles := Cycles;
END_METHOD

// Nothing to run. The run reports complete rather than waiting, so anything
// aggregating it is not held open.
METHOD Skip
IF NOT _IsOpen THEN
	RETURN;
END_IF

_IsOpen := FALSE;
_Tally.Begin(0);
_Index	:= TO_DINT(_Count);
THIS^.Finish();
END_METHOD

PROPERTY SkippedCount : UDINT
GET
SkippedCount := _Tally.SkippedCount;
END_GET
END_PROPERTY

// Suites the watchdog abandoned. Assert it is zero in CI: a stalled suite is never
// a normal outcome, and the run it belongs to cannot be trusted.
PROPERTY StalledSuites : UDINT
GET
StalledSuites := _StalledSuites;
END_GET
END_PROPERTY

// Suites added. Assert it in CI: a suite that silently stops being added takes
// its tests with it, and the totals simply come out smaller.
PROPERTY SuiteCount : UDINT
GET
SuiteCount := _Count;
END_GET
END_PROPERTY

PROPERTY TestCount : UDINT
GET
TestCount := _Tally.TestCount;
END_GET
END_PROPERTY

PROPERTY TotalDuration : LREAL
GET
TotalDuration := _Tally.TotalDuration;
END_GET
END_PROPERTY

END_FUNCTION_BLOCK

// ---- POUs/TestRunTally.TcPOU
// The counts, and what they add up to. The read model of a run.

//

// Separated from the suite because "what does this run amount to" is its own

// question, with its own consumers - CI, an HMI, a sequencer aggregating several -

// and none of them should be handed the ability to start or stop anything.

//

// Every figure is maintained INCREMENTALLY, as each test completes. Recomputing

// them by walking every slot each scan costs O(tests x capacity) every cycle, and

// still leaves nothing able to ask whether the run has finished.

//

// Not generic and holds nothing generic: it counts, and a count does not care how

// many slots exist.
FUNCTION_BLOCK TestRunTally IMPLEMENTS I_TestRunStatus
VAR
	_Status : ST_TestRunStatus;
END_VAR

(*
	No cyclic body. Figures change when a test finishes, not every scan.
*)

// Fold a whole nested result into these totals - one suite into a run, or one run

// into a larger one.

//

// Counts TESTS, not suites. A consumer polling the top of a nest wants to know

// how many tests passed, not how many containers did. Nesting is only worth having

// if the figures mean the same thing at every level.
METHOD Absorb
VAR_INPUT
	Status : I_TestRunStatus;
END_VAR
IF Status = 0 THEN
	RETURN;
END_IF

_Status.TestCount	  := _Status.TestCount + Status.TestCount;
_Status.PassedCount	  := _Status.PassedCount + Status.PassedCount;
_Status.FailedCount	  := _Status.FailedCount + Status.FailedCount;
_Status.ErrorCount	  := _Status.ErrorCount + Status.ErrorCount;
_Status.SkippedCount  := _Status.SkippedCount + Status.SkippedCount;
_Status.TotalDuration := _Status.TotalDuration + Status.TotalDuration;
END_METHOD

// Start a run over Count tests. Clears every figure but the label.

//

// Also what a re-run calls. A re-run re-executes the registered set, so the counts

// start again from nothing while the set itself is untouched.
METHOD Begin
VAR_INPUT
	Count : UDINT;
END_VAR
_Status.Outcome		  := E_RunOutcome.Running;
_Status.IsComplete	  := FALSE;
_Status.TestCount	  := Count;
_Status.PassedCount	  := 0;
_Status.FailedCount	  := 0;
_Status.ErrorCount	  := 0;
_Status.SkippedCount  := 0;
_Status.TotalDuration := 0.0;
END_METHOD

// Tests that could not run, plus framework errors.
PROPERTY ErrorCount : UDINT
GET
ErrorCount := _Status.ErrorCount;
END_GET
END_PROPERTY

// Checks that did not hold.
PROPERTY FailedCount : UDINT
GET
FailedCount := _Status.FailedCount;
END_GET
END_PROPERTY

// Terminal. Settles the aggregate outcome from what was recorded.

//

// Named Finish, not Complete: a status word as a method name reads as a question

// rather than an instruction, and

// Complete would sit beside the IsComplete property on this very object. That is

// exactly the collision the rule names.

//

// Aggregation, applied in order:

//   any Errored -> Errored   the run cannot be trusted

//   any Failed  -> Failed

//   all Skipped -> Skipped

//   otherwise   -> Passed

//

// Errored outranks Failed because a framework or environment problem casts doubt

// on every other result in the run. This is order-INSENSITIVE by design: a test

// that errored and then failed weighs the same as one that failed and then

// errored.
METHOD Finish
IF _Status.IsComplete THEN
	RETURN;
END_IF

IF _Status.ErrorCount > 0 THEN
	_Status.Outcome := E_RunOutcome.Errored;
ELSIF _Status.FailedCount > 0 THEN
	_Status.Outcome := E_RunOutcome.Failed;
ELSIF (_Status.SkippedCount > 0) AND (_Status.PassedCount = 0) THEN
	// Judged on TEST counts alone, which mean the same thing at every level of a
	// nest. Counting results folded in instead compared tests with suites once
	// Absorb was involved: a pass beside two skips in two suites settled as
	// Skipped, and a lone suite of two skips as Passed. Within a suite the two
	// rules agree, because there every result folded in is one test.
	_Status.Outcome := E_RunOutcome.Skipped;
ELSIF _Status.PassedCount > 0 THEN
	_Status.Outcome := E_RunOutcome.Passed;
ELSE
	// Nothing ran and nothing was skipped. An empty suite is a clean result, not a
	// failure - a project may legitimately deploy one with no tests registered.
	_Status.Outcome := E_RunOutcome.Passed;
END_IF

_Status.IsComplete := TRUE;
END_METHOD

// Reached a terminal state - NOT "ran everything".
PROPERTY IsComplete : BOOL
GET
IsComplete := _Status.IsComplete;
END_GET
END_PROPERTY

PROPERTY Label : T_MaxString
GET
Label := _Status.Label;
END_GET
END_PROPERTY

// Readable while the run is in progress: Running is distinct from every

// terminal value.
PROPERTY Outcome : E_RunOutcome
GET
Outcome := _Status.Outcome;
END_GET
END_PROPERTY

PROPERTY PassedCount : UDINT
GET
PassedCount := _Status.PassedCount;
END_GET
END_PROPERTY

// Fold one finished test into the totals.

//

// Called once per test as it completes, NOT recomputed every scan. Deriving the

// counts by walking every slot each cycle costs O(tests x capacity) and exposes

// none of the result anyway.

//

// A status that is not terminal is ignored rather than counted as something. There

// is no sensible bucket for Running, and inventing one would let a half-finished

// test look like a result.
METHOD Record
VAR_INPUT
	// Named Verdict, not Status: a parameter called Status would shadow the Status

	// property on this object, and the shadowing is silent.
	Verdict		: E_TestStatus;
	ElapsedTime : LREAL;
END_VAR
CASE Verdict OF
	E_TestStatus.Passed:
		_Status.PassedCount := _Status.PassedCount + 1;

	E_TestStatus.Failed:
		_Status.FailedCount := _Status.FailedCount + 1;

	E_TestStatus.Errored:
		_Status.ErrorCount := _Status.ErrorCount + 1;

	E_TestStatus.Skipped:
		_Status.SkippedCount := _Status.SkippedCount + 1;

ELSE
	RETURN;
END_CASE

_Status.TotalDuration := _Status.TotalDuration + ElapsedTime;
END_METHOD

// Something the framework itself could not do: a rejected registration, a

// teardown that overran, a result document that could not be written.

//

// It raises ErrorCount without touching TestCount, so the per-test figures still

// add up while the run is unmistakably untrustworthy. Reporting it as a test

// failure would send the reader hunting a defect that is not there.
METHOD RecordFrameworkError
_Status.ErrorCount := _Status.ErrorCount + 1;
END_METHOD

// The name this run reports under. Supplied by the suite at composition.
METHOD SetLabel
VAR_INPUT
	Label : T_MaxString;
END_VAR
_Status.Label := Label;
END_METHOD

// Not a failure. Must not turn a build red.
PROPERTY SkippedCount : UDINT
GET
SkippedCount := _Status.SkippedCount;
END_GET
END_PROPERTY

// Every figure at once, as a plain struct, for publishing as an ADS symbol.

//

// Copy it to a variable before reading a member: TwinCAT will not take a member

// off the result of a call.
PROPERTY Status : ST_TestRunStatus
GET
Status := _Status;
END_GET
END_PROPERTY

// Tests registered.
PROPERTY TestCount : UDINT
GET
TestCount := _Status.TestCount;
END_GET
END_PROPERTY

// Seconds for the whole run: a suite sums its tests, a sequencer sums its suites.

//

// Named apart from I_TestTiming.ElapsedTime deliberately - one is how long a

// single test has been going, the other an aggregate over many.
PROPERTY TotalDuration : LREAL
GET
TotalDuration := _Status.TotalDuration;
END_GET
END_PROPERTY

END_FUNCTION_BLOCK

// ---- POUs/TestReporterFanout.TcPOU
// One sink standing for many. A suite holds a single I_TestReporter and never

// learns how many are behind it.

//

// The composite is what makes several reporting problems disappear

// rather than get solved. The individual re-run that "records nothing and saves

// nothing" becomes a matter of NOT CALLING this object, rather than a flag

// threaded through the runner. Severity policy and the duplicated event-logger

// blocks become choices about which sinks a build attaches.

//

// It can also be SUSPENDED, which is what makes an individual re-run possible

// without a condition threaded through the runner.

//

// It implements I_TestDetailSink as well, and fans checks out only to the sinks

// that wanted them. Each reporter is queried once, when it is attached; a

// per-check query would put an interface lookup in the hottest path in the

// library.

//

// Not generic. Its capacity is a parameter rather than a generic argument because

// a project attaches the same set of sinks to every suite it owns, so per-instance

// variation would cost every declaration site an argument to buy nothing.
FUNCTION_BLOCK TestReporterFanout IMPLEMENTS I_TestReporter, I_TestDetailSink
VAR
	_Reporters : ARRAY[0..TestHarnessParameter.ReporterCapacity - 1] OF I_TestReporter;

	// Parallel to _Reporters: element i is the detail face of reporter i, or null

	// where that reporter did not want checks. Resolved once, at Add.
	_DetailSinks : ARRAY[0..TestHarnessParameter.ReporterCapacity - 1] OF I_TestDetailSink;
	_Count		 : UDINT;

	// While TRUE, notifications are dropped and nothing reaches a sink.

	//

	// This is how an individual re-run records nothing and saves nothing: the suite

	// silences every sink at once, rather than a condition threaded through the

	// runner and the journal and remembered in three places.

	//

	// CyclicLogic is NOT suppressed. A file write already in flight must still

	// finish, or IsIdle never goes TRUE and CI waits forever.
	_IsSuspended : BOOL;
END_VAR

(*
	No cyclic body of its own. CyclicLogic is the cyclic entry point and is called
	by the suite, which is itself driven.
*)

// Attach a sink. Order of attachment is order of notification.

//

// Not named Add: ADD is a standard function and TwinCAT is case-insensitive.

//

// Every reporter attached receives everything; there is no filtering here, because

// a sink that wants less can decide that for itself.

//

// A reporter is queried ONCE for I_TestDetailSink and the answer is stored. A

// per-check __QUERYINTERFACE would put an interface lookup inside the hottest path

// in the library - a forty-check test would pay for forty of them.

//

// Returns FALSE when the list is full or the reporter is null, and raises a

// framework error through the sinks ALREADY attached. That is not circular: the

// ones already there are exactly the ones that can still report it.
METHOD Attach : BOOL
VAR_INPUT
	Reporter : I_TestReporter;
END_VAR

VAR
	Index : DINT;
END_VAR
Attach := FALSE;
IF Reporter = 0 THEN
	THIS^.FrameworkError('TestReporterFanout', 'a null reporter was offered');
	RETURN;
END_IF

IF _Count >= TestHarnessParameter.ReporterCapacity THEN
	THIS^.FrameworkError('TestReporterFanout', 'reporter list is full - raise TestHarnessParameter.ReporterCapacity');
	RETURN;
END_IF

Index			  := TO_DINT(_Count);
_Reporters[Index] := Reporter;
// Optional, exactly as the test hooks are. A sink that only wants verdicts does

// not implement it and is never called for checks.
IF NOT __QUERYINTERFACE(Reporter, _DetailSinks[Index]) THEN
	_DetailSinks[Index] := 0;
END_IF

_Count := _Count + 1;
Attach := TRUE;
END_METHOD

METHOD CheckFailed
VAR_INPUT
	StepLabel  : T_MaxString;
	Kind	   : E_FailureKind;
	Expected   : T_MaxString;
	Actual	   : T_MaxString;
	Diagnostic : T_MaxString;
	Message	   : T_MaxString;
END_VAR

VAR
	i : DINT;
END_VAR
IF _IsSuspended THEN
	RETURN;
END_IF

FOR i := 0 TO TO_DINT(_Count) - 1 DO
	IF _DetailSinks[i] <> 0 THEN
		_DetailSinks[i].CheckFailed(StepLabel  := StepLabel,
									Kind	   := Kind,
									Expected   := Expected,
									Actual	   := Actual,
									Diagnostic := Diagnostic,
									Message	   := Message);
	END_IF
END_FOR
END_METHOD

METHOD CheckPassed
VAR_INPUT
	StepLabel : T_MaxString;
	Detail	  : T_MaxString;
END_VAR

VAR
	i : DINT;
END_VAR
IF _IsSuspended THEN
	RETURN;
END_IF

FOR i := 0 TO TO_DINT(_Count) - 1 DO
	IF _DetailSinks[i] <> 0 THEN
		_DetailSinks[i].CheckPassed(StepLabel := StepLabel, Detail := Detail);
	END_IF
END_FOR
END_METHOD

// Sinks attached. Assert it in CI: a reporter that silently stops being attached

// takes its output with it, and a result file that never appears reads as a broken

// build rather than as a missing sink.
PROPERTY Count : UDINT
GET
Count := _Count;
END_GET
END_PROPERTY

// Advance every sink, every scan, unconditionally.

//

